   DATA[942,18] := 1.0;
   DATA[942,19] := 1.0;
   DATA[942,20] := 148.808;
   DATA[942,21] := 155.0628;
   DATA[942,22] := 1.71608;
   DATA[942,23] := 928.262;
   DATA[942,24] := 2.0;
   DATA[942,25] := 2.0;
   DATA[942,26] := 7.87798;
   DATA[942,27] := 144.3989;
   DATA[942,28] := 263.0415;
   DATA[942,29] := 11.95847;
   DATA[942,30] := 1.726096;
   DATA[942,31] := 1.281542;
   DATA[942,32] := 0.7357808;
   DATA[942,33] := 0.306761;
   DATA[942,34] := 2.0;
   DATA[942,35] := 250.7049;
   DATA[942,36] := 1.746067;
   DATA[942,37] := 189.5187;
   DATA[942,38] := 0.000128152;
   DATA[942,39] := 1.0;
   DATA[943,0] := 2.542356;
   DATA[943,1] := 627.6909;
   DATA[943,2] := 2.0;
   DATA[943,3] := 1.0;
   DATA[943,4] := 262.4648;
   DATA[943,5] := 8.460844;
   DATA[943,6] := 315.4576;
   DATA[943,8] := 1.0;
   DATA[943,9] := 1.0;
   DATA[943,10] := 1.0;
   DATA[943,11] := 2.010372;
   DATA[943,13] := 1010.839;
   DATA[943,14] := 1.0;
   DATA[943,15] := 1.0;
   DATA[943,16] := 1.0;
   DATA[943,17] := 1.0;
   DATA[943,18] := 1.0;
   DATA[943,19] := 1.0;
   DATA[943,20] := 148.808;
   DATA[943,21] := 155.0628;
   DATA[943,22] := 1.71608;
   DATA[943,23] := 928.1466;
   DATA[943,24] := 2.0;
   DATA[943,25] := 2.0;
   DATA[943,26] := 7.87798;
   DATA[943,27] := 144.3989;
   DATA[943,28] := 263.0415;
   DATA[943,29] := 11.95847;
   DATA[943,30] := 1.726096;
   DATA[943,31] := 1.287306;
   DATA[943,32] := 0.7357808;
   DATA[943,33] := 0.3070813;
   DATA[943,34] := 2.0;
   DATA[943,35] := 250.7049;
   DATA[943,36] := 1.746067;
   DATA[943,37] := 189.5187;
   DATA[943,38] := 0.000128152;
   DATA[943,39] := 1.0;
   DATA[944,0] := 2.540435;
   DATA[944,1] := 627.6124;
   DATA[944,2] := 2.0;
   DATA[944,3] := 1.0;
   DATA[944,4] := 262.4648;
   DATA[944,5] := 8.460844;
   DATA[944,6] := 315.4576;
   DATA[944,8] := 1.0;
   DATA[944,9] := 1.0;
   DATA[944,10] := 1.0;
   DATA[944,11] := 2.010372;
   DATA[944,13] := 1010.718;
   DATA[944,14] := 1.0;
   DATA[944,15] := 1.0;
   DATA[944,16] := 1.0;
   DATA[944,17] := 1.0;
   DATA[944,18] := 1.0;
   DATA[944,19] := 1.0;
   DATA[944,20] := 148.808;
   DATA[944,21] := 155.0628;
   DATA[944,22] := 1.717489;
   DATA[944,23] := 928.1466;
   DATA[944,24] := 2.0;
   DATA[944,25] := 2.0;
   DATA[944,26] := 7.87798;
   DATA[944,27] := 144.3989;
   DATA[944,28] := 263.0415;
   DATA[944,29] := 11.95847;
   DATA[944,30] := 1.728659;
   DATA[944,31] := 1.290893;
   DATA[944,32] := 0.7357808;
   DATA[944,33] := 0.3070813;
   DATA[944,34] := 2.0;
   DATA[944,35] := 250.7049;
   DATA[944,36] := 1.746067;
   DATA[944,37] := 189.5187;
   DATA[944,38] := 0.000128152;
   DATA[944,39] := 1.0;
   DATA[945,0] := 2.540435;
   DATA[945,1] := 627.8086;
   DATA[945,2] := 2.0;
   DATA[945,3] := 1.0;
   DATA[945,4] := 262.4648;
   DATA[945,5] := 8.460844;
   DATA[945,6] := 315.4576;
   DATA[945,8] := 1.0;
   DATA[945,9] := 1.0;
   DATA[945,10] := 1.0;
   DATA[945,11] := 2.010372;
   DATA[945,13] := 1010.959;
   DATA[945,14] := 1.0;
   DATA[945,15] := 1.0;
   DATA[945,16] := 1.0;
   DATA[945,17] := 1.0;
   DATA[945,18] := 1.0;
   DATA[945,19] := 1.0;
   DATA[945,20] := 148.808;
   DATA[945,21] := 155.0628;
   DATA[945,22] := 1.717489;
   DATA[945,23] := 928.1466;
   DATA[945,24] := 2.0;
   DATA[945,25] := 2.0;
   DATA[945,26] := 7.87798;
   DATA[945,27] := 144.3989;
   DATA[945,28] := 263.0415;
   DATA[945,29] := 11.95847;
   DATA[945,30] := 1.728659;
   DATA[945,31] := 1.271551;
   DATA[945,32] := 0.7357808;
   DATA[945,33] := 0.3070813;
   DATA[945,34] := 2.0;
   DATA[945,35] := 250.7049;
   DATA[945,36] := 1.746067;
   DATA[945,37] := 189.5187;
   DATA[945,38] := 0.000128152;
   DATA[945,39] := 1.0;
   DATA[946,0] := 2.540435;
   DATA[946,1] := 628.4366;
   DATA[946,2] := 2.0;
   DATA[946,3] := 1.0;
   DATA[946,4] := 262.4648;
   DATA[946,5] := 8.460844;
   DATA[946,6] := 315.4576;
   DATA[946,8] := 1.0;
   DATA[946,9] := 1.0;
   DATA[946,10] := 1.0;
   DATA[946,11] := 2.010372;
   DATA[946,13] := 1010.638;
   DATA[946,14] := 1.0;
   DATA[946,15] := 1.0;
   DATA[946,16] := 1.0;
   DATA[946,17] := 1.0;
   DATA[946,18] := 1.0;
   DATA[946,19] := 1.0;
   DATA[946,20] := 148.808;
   DATA[946,21] := 155.0628;
   DATA[946,22] := 1.717489;
   DATA[946,23] := 927.8005;
   DATA[946,24] := 2.0;
   DATA[946,25] := 2.0;
   DATA[946,26] := 7.87798;
   DATA[946,27] := 144.3989;
   DATA[946,28] := 263.0415;
   DATA[946,29] := 12.07383;
   DATA[946,30] := 1.728659;
   DATA[946,31] := 1.265275;
   DATA[946,32] := 0.7348846;
   DATA[946,33] := 0.3066329;
   DATA[946,34] := 2.0;
   DATA[946,35] := 250.5608;
   DATA[946,36] := 1.746067;
   DATA[946,37] := 189.5187;
   DATA[946,38] := 0.000128152;
   DATA[946,39] := 1.0;
   DATA[947,0] := 2.545239;
   DATA[947,1] := 629.3395;
   DATA[947,2] := 2.0;
   DATA[947,3] := 1.0;
   DATA[947,4] := 262.4648;
   DATA[947,5] := 8.460844;
   DATA[947,6] := 315.4576;
   DATA[947,8] := 1.0;
   DATA[947,9] := 1.0;
   DATA[947,10] := 1.0;
   DATA[947,11] := 2.010372;
   DATA[947,13] := 1011.119;
   DATA[947,14] := 1.0;
   DATA[947,15] := 1.0;
   DATA[947,16] := 1.0;
   DATA[947,17] := 1.0;
   DATA[947,18] := 1.0;
   DATA[947,19] := 1.0;
   DATA[947,20] := 148.808;
   DATA[947,21] := 155.0628;
   DATA[947,22] := 1.717489;
   DATA[947,23] := 927.3007;
   DATA[947,24] := 2.0;
   DATA[947,25] := 2.0;
   DATA[947,26] := 7.87798;
   DATA[947,27] := 144.3989;
   DATA[947,28] := 263.0415;
   DATA[947,29] := 12.07383;
   DATA[947,30] := 1.728659;
   DATA[947,31] := 1.267196;
   DATA[947,32] := 0.7348846;
   DATA[947,33] := 0.3066329;
   DATA[947,34] := 2.0;
   DATA[947,35] := 250.5447;
   DATA[947,36] := 1.746067;
   DATA[947,37] := 189.5187;
   DATA[947,38] := 0.000128152;
   DATA[947,39] := 1.0;
   DATA[948,0] := 2.552926;
   DATA[948,1] := 630.1245;
   DATA[948,2] := 2.0;
   DATA[948,3] := 1.0;
   DATA[948,4] := 262.4648;
   DATA[948,5] := 8.460844;
   DATA[948,6] := 315.4576;
   DATA[948,8] := 1.0;
   DATA[948,9] := 1.0;
   DATA[948,10] := 1.0;
   DATA[948,11] := 2.010372;
   DATA[948,13] := 1010.638;
   DATA[948,14] := 1.0;
   DATA[948,15] := 1.0;
   DATA[948,16] := 1.0;
   DATA[948,17] := 1.0;
   DATA[948,18] := 1.0;
   DATA[948,19] := 1.0;
   DATA[948,20] := 148.808;
   DATA[948,21] := 155.0628;
   DATA[948,22] := 1.717489;
   DATA[948,23] := 927.1085;
   DATA[948,24] := 2.0;
   DATA[948,25] := 2.0;
   DATA[948,26] := 7.87798;
   DATA[948,27] := 144.3989;
   DATA[948,28] := 263.0415;
   DATA[948,29] := 12.07383;
   DATA[948,30] := 1.728659;
   DATA[948,31] := 1.261176;
   DATA[948,32] := 0.7348846;
   DATA[948,33] := 0.3066329;
   DATA[948,34] := 2.0;
   DATA[948,35] := 250.5447;
   DATA[948,36] := 1.746067;
   DATA[948,37] := 189.3585;
   DATA[948,38] := 0.000128152;
   DATA[948,39] := 1.0;
   DATA[949,0] := 2.55773;
   DATA[949,1] := 631.3414;
   DATA[949,2] := 2.0;
   DATA[949,3] := 1.0;
   DATA[949,4] := 262.4648;
   DATA[949,5] := 8.460844;
   DATA[949,6] := 315.4576;
   DATA[949,8] := 1.0;
   DATA[949,9] := 1.0;
   DATA[949,10] := 1.0;
   DATA[949,11] := 2.010372;
   DATA[949,13] := 1011.159;
   DATA[949,14] := 1.0;
   DATA[949,15] := 1.0;
   DATA[949,16] := 1.0;
   DATA[949,17] := 1.0;
   DATA[949,18] := 1.0;
   DATA[949,19] := 1.0;
   DATA[949,20] := 148.808;
   DATA[949,21] := 155.0628;
   DATA[949,22] := 1.717489;
   DATA[949,23] := 927.3007;
   DATA[949,24] := 2.0;
   DATA[949,25] := 2.0;
   DATA[949,26] := 7.87798;
   DATA[949,27] := 144.3989;
   DATA[949,28] := 263.0415;
   DATA[949,29] := 12.07383;
   DATA[949,30] := 1.728659;
   DATA[949,31] := 1.265659;
   DATA[949,32] := 0.7348846;
   DATA[949,33] := 0.3066329;
   DATA[949,34] := 2.0;
   DATA[949,35] := 250.5447;
   DATA[949,36] := 1.746067;
   DATA[949,37] := 189.3585;
   DATA[949,38] := 0.000128152;
   DATA[949,39] := 1.0;
   DATA[950,0] := 2.55773;
   DATA[950,1] := 632.3619;
   DATA[950,2] := 2.0;
   DATA[950,3] := 1.0;
   DATA[950,4] := 262.4648;
   DATA[950,5] := 8.460844;
   DATA[950,6] := 315.5089;
   DATA[950,8] := 1.0;
   DATA[950,9] := 1.0;
   DATA[950,10] := 1.0;
   DATA[950,11] := 2.010372;
   DATA[950,13] := 1011.119;
   DATA[950,14] := 1.0;
   DATA[950,15] := 1.0;
   DATA[950,16] := 1.0;
   DATA[950,17] := 1.0;
   DATA[950,18] := 1.0;
   DATA[950,19] := 1.0;
   DATA[950,20] := 148.808;
   DATA[950,21] := 155.0628;
   DATA[950,22] := 1.717489;
   DATA[950,23] := 927.2238;
   DATA[950,24] := 2.0;
   DATA[950,25] := 2.0;
   DATA[950,26] := 7.87798;
   DATA[950,27] := 144.3989;
   DATA[950,28] := 263.0415;
   DATA[950,29] := 12.07383;
   DATA[950,30] := 1.728659;
   DATA[950,31] := 1.280517;
   DATA[950,32] := 0.7348846;
   DATA[950,33] := 0.3066329;
   DATA[950,34] := 2.0;
   DATA[950,35] := 250.5447;
   DATA[950,36] := 1.746067;
   DATA[950,37] := 189.3585;
   DATA[950,38] := 0.000128152;
   DATA[950,39] := 1.0;
   DATA[951,0] := 2.55773;
   DATA[951,1] := 633.3825;
   DATA[951,2] := 2.0;
   DATA[951,3] := 1.0;
   DATA[951,4] := 262.4648;
   DATA[951,5] := 8.460844;
   DATA[951,6] := 315.5601;
   DATA[951,8] := 1.0;
   DATA[951,9] := 1.0;
   DATA[951,10] := 1.0;
   DATA[951,11] := 2.010372;
   DATA[951,13] := 1010.758;
   DATA[951,14] := 1.0;
   DATA[951,15] := 1.0;
   DATA[951,16] := 1.0;
   DATA[951,17] := 1.0;
   DATA[951,18] := 1.0;
   DATA[951,19] := 1.0;
   DATA[951,20] := 148.808;
   DATA[951,21] := 155.2166;
   DATA[951,22] := 1.717489;
   DATA[951,23] := 926.6086;
   DATA[951,24] := 2.0;
   DATA[951,25] := 2.0;
   DATA[951,26] := 7.87798;
   DATA[951,27] := 144.3989;
   DATA[951,28] := 263.0415;
   DATA[951,29] := 12.07383;
   DATA[951,30] := 1.726865;
   DATA[951,31] := 1.291405;
   DATA[951,32] := 0.7348846;
   DATA[951,33] := 0.3066329;
   DATA[951,34] := 2.0;
   DATA[951,35] := 250.4166;
   DATA[951,36] := 1.69801;
   DATA[951,37] := 189.2464;
   DATA[951,38] := 0.000128152;
   DATA[951,39] := 1.0;
   DATA[952,0] := 2.556129;
   DATA[952,1] := 634.1675;
   DATA[952,2] := 2.0;
   DATA[952,3] := 1.0;
   DATA[952,4] := 262.4648;
   DATA[952,5] := 8.460844;
   DATA[952,6] := 315.5601;
   DATA[952,8] := 1.0;
   DATA[952,9] := 1.0;
   DATA[952,10] := 1.0;
   DATA[952,11] := 2.010372;
   DATA[952,13] := 1010.879;
   DATA[952,14] := 1.0;
   DATA[952,15] := 1.0;
   DATA[952,16] := 1.0;
   DATA[952,17] := 1.0;
   DATA[952,18] := 1.0;
   DATA[952,19] := 1.0;
   DATA[952,20] := 148.808;
   DATA[952,21] := 155.2166;
   DATA[952,22] := 1.717489;
   DATA[952,23] := 926.0703;
   DATA[952,24] := 2.0;
   DATA[952,25] := 2.0;
   DATA[952,26] := 7.87798;
   DATA[952,27] := 144.3989;
   DATA[952,28] := 263.0415;
   DATA[952,29] := 12.07383;
   DATA[952,30] := 1.726865;
   DATA[952,31] := 1.300884;
   DATA[952,32] := 0.7348846;
   DATA[952,33] := 0.3072094;
   DATA[952,34] := 2.0;
   DATA[952,35] := 250.4166;
   DATA[952,36] := 1.69801;
   DATA[952,37] := 189.2464;
   DATA[952,38] := 0.000128152;
   DATA[952,39] := 1.0;
   DATA[953,0] := 2.547161;
   DATA[953,1] := 635.2667;
   DATA[953,2] := 2.0;
   DATA[953,3] := 1.0;
   DATA[953,4] := 262.4648;
   DATA[953,5] := 8.460844;
   DATA[953,6] := 315.5601;
   DATA[953,8] := 1.0;
   DATA[953,9] := 1.0;
   DATA[953,10] := 1.0;
   DATA[953,11] := 2.010372;
   DATA[953,13] := 1011.079;
   DATA[953,14] := 1.0;
   DATA[953,15] := 1.0;
   DATA[953,16] := 1.0;
   DATA[953,17] := 1.0;
   DATA[953,18] := 1.0;
   DATA[953,19] := 1.0;
   DATA[953,20] := 148.808;
   DATA[953,21] := 155.2166;
   DATA[953,22] := 1.717489;
   DATA[953,23] := 925.6857;
   DATA[953,24] := 2.0;
   DATA[953,25] := 2.0;
   DATA[953,26] := 7.87798;
   DATA[953,27] := 144.3989;
   DATA[953,28] := 263.0415;
   DATA[953,29] := 12.07383;
   DATA[953,30] := 1.726737;
   DATA[953,31] := 1.300243;
   DATA[953,32] := 0.7348846;
   DATA[953,33] := 0.30785;
   DATA[953,34] := 2.0;
   DATA[953,35] := 250.4166;
   DATA[953,36] := 1.69801;
   DATA[953,37] := 189.2464;
   DATA[953,38] := 0.000128152;
   DATA[953,39] := 1.0;
   DATA[954,0] := 2.547161;
   DATA[954,1] := 635.2274;
   DATA[954,2] := 2.0;
   DATA[954,3] := 1.0;
   DATA[954,4] := 262.4648;
   DATA[954,5] := 8.460844;
   DATA[954,6] := 315.6114;
   DATA[954,8] := 1.0;
   DATA[954,9] := 1.0;
   DATA[954,10] := 1.0;
   DATA[954,11] := 2.010372;
   DATA[954,13] := 1010.758;
   DATA[954,14] := 1.0;
   DATA[954,15] := 1.0;
   DATA[954,16] := 1.0;
   DATA[954,17] := 1.0;
   DATA[954,18] := 1.0;
   DATA[954,19] := 1.0;
   DATA[954,20] := 148.808;
   DATA[954,21] := 155.0115;
   DATA[954,22] := 1.717489;
   DATA[954,23] := 925.7626;
   DATA[954,24] := 2.0;
   DATA[954,25] := 2.0;
   DATA[954,26] := 7.87798;
   DATA[954,27] := 144.3989;
   DATA[954,28] := 263.0415;
   DATA[954,29] := 12.07383;
   DATA[954,30] := 1.725968;
   DATA[954,31] := 1.292174;
   DATA[954,32] := 0.7348846;
   DATA[954,33] := 0.3084905;
   DATA[954,34] := 2.0;
   DATA[954,35] := 250.4005;
   DATA[954,36] := 1.69801;
   DATA[954,37] := 189.2464;
   DATA[954,38] := 0.000128152;
   DATA[954,39] := 1.0;
   DATA[955,0] := 2.542677;
   DATA[955,1] := 636.2872;
   DATA[955,2] := 2.0;
   DATA[955,3] := 1.0;
   DATA[955,4] := 262.4648;
   DATA[955,5] := 8.460844;
   DATA[955,6] := 315.6114;
   DATA[955,8] := 1.0;
   DATA[955,9] := 1.0;
   DATA[955,10] := 1.0;
   DATA[955,11] := 2.010372;
   DATA[955,13] := 1010.758;
   DATA[955,14] := 1.0;
   DATA[955,15] := 1.0;
   DATA[955,16] := 1.0;
   DATA[955,17] := 1.0;
   DATA[955,18] := 1.0;
   DATA[955,19] := 1.0;
   DATA[955,20] := 148.808;
   DATA[955,21] := 155.0115;
   DATA[955,22] := 1.717489;
   DATA[955,23] := 925.0705;
   DATA[955,24] := 2.0;
   DATA[955,25] := 2.0;
   DATA[955,26] := 7.87798;
   DATA[955,27] := 144.3989;
   DATA[955,28] := 263.0415;
   DATA[955,29] := 12.07383;
   DATA[955,30] := 1.725583;
   DATA[955,31] := 1.292174;
   DATA[955,32] := 0.7357808;
   DATA[955,33] := 0.3084905;
   DATA[955,34] := 2.0;
   DATA[955,35] := 250.4005;
   DATA[955,36] := 1.69801;
   DATA[955,37] := 189.2464;
   DATA[955,38] := 0.000128152;
   DATA[955,39] := 1.0;
   DATA[956,0] := 2.542677;
   DATA[956,1] := 636.6013;
   DATA[956,2] := 2.0;
   DATA[956,3] := 1.0;
   DATA[956,4] := 262.4648;
   DATA[956,5] := 8.460844;
   DATA[956,6] := 315.6114;
   DATA[956,8] := 1.0;
   DATA[956,9] := 1.0;
   DATA[956,10] := 1.0;
   DATA[956,11] := 2.010372;
   DATA[956,13] := 1010.919;
   DATA[956,14] := 1.0;
   DATA[956,15] := 1.0;
   DATA[956,16] := 1.0;
   DATA[956,17] := 1.0;
   DATA[956,18] := 1.0;
   DATA[956,19] := 1.0;
   DATA[956,20] := 148.808;
   DATA[956,21] := 155.0115;
   DATA[956,22] := 1.714542;
   DATA[956,23] := 924.6475;
   DATA[956,24] := 2.0;
   DATA[956,25] := 2.0;
   DATA[956,26] := 7.87798;
   DATA[956,27] := 144.3989;
   DATA[956,28] := 263.0415;
   DATA[956,29] := 12.07383;
   DATA[956,30] := 1.725583;
   DATA[956,31] := 1.296273;
   DATA[956,32] := 0.7357808;
   DATA[956,33] := 0.3084905;
   DATA[956,34] := 2.0;
   DATA[956,35] := 250.4005;
   DATA[956,36] := 1.69801;
   DATA[956,37] := 189.2464;
   DATA[956,38] := 0.000128152;
   DATA[956,39] := 1.0;
   DATA[957,0] := 2.542677;
   DATA[957,1] := 637.2686;
   DATA[957,2] := 2.0;
   DATA[957,3] := 1.0;
   DATA[957,4] := 262.4648;
   DATA[957,5] := 8.460844;
   DATA[957,6] := 315.6114;
   DATA[957,8] := 1.0;
   DATA[957,9] := 1.0;
   DATA[957,10] := 1.0;
   DATA[957,11] := 2.010372;
   DATA[957,13] := 1010.718;
   DATA[957,14] := 1.0;
   DATA[957,15] := 1.0;
   DATA[957,16] := 1.0;
   DATA[957,17] := 1.0;
   DATA[957,18] := 1.0;
   DATA[957,19] := 1.0;
   DATA[957,20] := 148.808;
   DATA[957,21] := 155.2166;
   DATA[957,22] := 1.714542;
   DATA[957,23] := 924.0707;
   DATA[957,24] := 2.0;
   DATA[957,25] := 2.0;
   DATA[957,26] := 7.87798;
   DATA[957,27] := 144.3989;
   DATA[957,28] := 263.0415;
   DATA[957,29] := 12.07383;
   DATA[957,30] := 1.724045;
   DATA[957,31] := 1.302677;
   DATA[957,32] := 0.7357808;
   DATA[957,33] := 0.3084905;
   DATA[957,34] := 2.0;
   DATA[957,35] := 250.4005;
   DATA[957,36] := 1.69801;
   DATA[957,37] := 189.2464;
   DATA[957,38] := 0.000128152;
   DATA[957,39] := 1.0;
   DATA[958,0] := 2.550364;
   DATA[958,1] := 637.5825;
   DATA[958,2] := 2.0;
   DATA[958,3] := 1.0;
   DATA[958,4] := 262.4648;
   DATA[958,5] := 8.460844;
   DATA[958,6] := 315.6114;
   DATA[958,8] := 1.0;
   DATA[958,9] := 1.0;
   DATA[958,10] := 1.0;
   DATA[958,11] := 2.010372;
   DATA[958,13] := 1010.518;
   DATA[958,14] := 1.0;
   DATA[958,15] := 1.0;
   DATA[958,16] := 1.0;
   DATA[958,17] := 1.0;
   DATA[958,18] := 1.0;
   DATA[958,19] := 1.0;
   DATA[958,20] := 148.808;
   DATA[958,21] := 155.2166;
   DATA[958,22] := 1.714542;
   DATA[958,23] := 923.5709;
   DATA[958,24] := 2.0;
   DATA[958,25] := 2.0;
   DATA[958,26] := 7.87798;
   DATA[958,27] := 144.3989;
   DATA[958,28] := 263.0415;
   DATA[958,29] := 12.07383;
   DATA[958,30] := 1.724045;
   DATA[958,31] := 1.302677;
   DATA[958,32] := 0.7357808;
   DATA[958,33] := 0.3084905;
   DATA[958,34] := 2.0;
   DATA[958,35] := 250.4005;
   DATA[958,36] := 1.69801;
   DATA[958,37] := 189.2464;
   DATA[958,38] := 0.000128152;
   DATA[958,39] := 1.0;
   DATA[959,0] := 2.552285;
   DATA[959,1] := 638.6031;
   DATA[959,2] := 2.0;
   DATA[959,3] := 1.0;
   DATA[959,4] := 262.4648;
   DATA[959,5] := 8.460844;
   DATA[959,6] := 315.6114;
   DATA[959,8] := 1.0;
   DATA[959,9] := 1.0;
   DATA[959,10] := 1.0;
   DATA[959,11] := 2.010372;
   DATA[959,13] := 1010.678;
   DATA[959,14] := 1.0;
   DATA[959,15] := 1.0;
   DATA[959,16] := 1.0;
   DATA[959,17] := 1.0;
   DATA[959,18] := 1.0;
   DATA[959,19] := 1.0;
   DATA[959,20] := 148.808;
   DATA[959,21] := 155.2166;
   DATA[959,22] := 1.715183;
   DATA[959,23] := 923.1479;
   DATA[959,24] := 2.0;
   DATA[959,25] := 2.0;
   DATA[959,26] := 7.87798;
   DATA[959,27] := 144.3989;
   DATA[959,28] := 263.0415;
   DATA[959,29] := 12.07383;
   DATA[959,30] := 1.724045;
   DATA[959,31] := 1.295376;
   DATA[959,32] := 0.7380853;
   DATA[959,33] := 0.3084905;
   DATA[959,34] := 2.0;
   DATA[959,35] := 250.4005;
   DATA[959,36] := 1.69801;
   DATA[959,37] := 189.2464;
   DATA[959,38] := 0.000128152;
   DATA[959,39] := 1.0;
   DATA[960,0] := 2.552285;
   DATA[960,1] := 639.5452;
   DATA[960,2] := 2.0;
   DATA[960,3] := 1.0;
   DATA[960,4] := 262.4648;
   DATA[960,5] := 8.460844;
   DATA[960,6] := 315.6114;
   DATA[960,8] := 1.0;
   DATA[960,9] := 1.0;
   DATA[960,10] := 1.0;
   DATA[960,11] := 2.010372;
   DATA[960,13] := 1010.839;
   DATA[960,14] := 1.0;
   DATA[960,15] := 1.0;
   DATA[960,16] := 1.0;
   DATA[960,17] := 1.0;
   DATA[960,18] := 1.0;
   DATA[960,19] := 1.0;
   DATA[960,20] := 148.808;
   DATA[960,21] := 155.2166;
   DATA[960,22] := 1.71608;
   DATA[960,23] := 922.9941;
   DATA[960,24] := 2.0;
   DATA[960,25] := 2.0;
   DATA[960,26] := 7.87798;
   DATA[960,27] := 144.3989;
   DATA[960,28] := 263.0415;
   DATA[960,29] := 12.07383;
   DATA[960,30] := 1.724045;
   DATA[960,31] := 1.283079;
   DATA[960,32] := 0.7380853;
   DATA[960,33] := 0.3084905;
   DATA[960,34] := 2.0;
   DATA[960,35] := 250.4005;
   DATA[960,36] := 1.69801;
   DATA[960,37] := 189.2464;
   DATA[960,38] := 0.000128152;
   DATA[960,39] := 1.0;
   DATA[961,0] := 2.552285;
   DATA[961,1] := 639.8592;
   DATA[961,2] := 2.0;
   DATA[961,3] := 1.0;
   DATA[961,4] := 262.4648;
   DATA[961,5] := 8.460844;
   DATA[961,6] := 315.6114;
   DATA[961,8] := 1.0;
   DATA[961,9] := 1.0;
   DATA[961,10] := 1.0;
   DATA[961,11] := 2.010372;
   DATA[961,13] := 1011.079;
   DATA[961,14] := 1.0;
   DATA[961,15] := 1.0;
   DATA[961,16] := 1.0;
   DATA[961,17] := 1.0;
   DATA[961,18] := 1.0;
   DATA[961,19] := 1.0;
   DATA[961,20] := 148.808;
   DATA[961,21] := 155.2166;
   DATA[961,22] := 1.71608;
   DATA[961,23] := 922.9172;
   DATA[961,24] := 2.0;
   DATA[961,25] := 2.0;
   DATA[961,26] := 7.87798;
   DATA[961,27] := 144.3989;
   DATA[961,28] := 263.0415;
   DATA[961,29] := 12.07383;
   DATA[961,30] := 1.724045;
   DATA[961,31] := 1.285513;
   DATA[961,32] := 0.7380853;
   DATA[961,33] := 0.3084905;
   DATA[961,34] := 2.0;
   DATA[961,35] := 250.1122;
   DATA[961,36] := 1.746067;
   DATA[961,37] := 189.1022;
   DATA[961,38] := 0.000128152;
   DATA[961,39] := 1.0;
   DATA[962,0] := 2.548762;
   DATA[962,1] := 640.5265;
   DATA[962,2] := 2.0;
   DATA[962,3] := 1.0;
   DATA[962,4] := 262.4648;
   DATA[962,5] := 8.460844;
   DATA[962,6] := 315.6114;
   DATA[962,8] := 1.0;
   DATA[962,9] := 1.0;
   DATA[962,10] := 1.0;
   DATA[962,11] := 2.010372;
   DATA[962,13] := 1010.758;
   DATA[962,14] := 1.0;
   DATA[962,15] := 1.0;
   DATA[962,16] := 1.0;
   DATA[962,17] := 1.0;
   DATA[962,18] := 1.0;
   DATA[962,19] := 1.0;
   DATA[962,20] := 148.808;
   DATA[962,21] := 155.2166;
   DATA[962,22] := 1.714798;
   DATA[962,23] := 922.6096;
   DATA[962,24] := 2.0;
   DATA[962,25] := 2.0;
   DATA[962,26] := 7.87798;
   DATA[962,27] := 144.3989;
   DATA[962,28] := 263.0415;
   DATA[962,29] := 12.07383;
   DATA[962,30] := 1.724045;
   DATA[962,31] := 1.291918;
   DATA[962,32] := 0.7380853;
   DATA[962,33] := 0.3084905;
   DATA[962,34] := 2.0;
   DATA[962,35] := 250.1122;
   DATA[962,36] := 1.762086;
   DATA[962,37] := 189.1022;
   DATA[962,38] := 0.000128152;
   DATA[962,39] := 1.0;
   DATA[963,0] := 2.543317;
   DATA[963,1] := 641.233;
   DATA[963,2] := 2.0;
   DATA[963,3] := 1.0;
   DATA[963,4] := 262.4648;
   DATA[963,5] := 8.462767;
   DATA[963,6] := 315.6114;
   DATA[963,8] := 1.0;
   DATA[963,9] := 1.0;
   DATA[963,10] := 1.0;
   DATA[963,11] := 2.010372;
   DATA[963,13] := 1010.919;
   DATA[963,14] := 1.0;
   DATA[963,15] := 1.0;
   DATA[963,16] := 1.0;
   DATA[963,17] := 1.0;
   DATA[963,18] := 1.0;
   DATA[963,19] := 1.0;
   DATA[963,20] := 148.808;
   DATA[963,21] := 155.1653;
   DATA[963,22] := 1.713261;
   DATA[963,23] := 922.6865;
   DATA[963,24] := 2.0;
   DATA[963,25] := 2.0;
   DATA[963,26] := 7.87798;
   DATA[963,27] := 144.3989;
   DATA[963,28] := 263.0415;
   DATA[963,29] := 12.07383;
   DATA[963,30] := 1.724045;
   DATA[963,31] := 1.30985;
   DATA[963,32] := 0.7380853;
   DATA[963,33] := 0.3084905;
   DATA[963,34] := 2.0;
   DATA[963,35] := 250.1122;
   DATA[963,36] := 1.762086;
   DATA[963,37] := 189.1022;
   DATA[963,38] := 0.000128152;
   DATA[963,39] := 1.0;
   DATA[964,0] := 2.540435;
   DATA[964,1] := 641.5863;
   DATA[964,2] := 2.0;
   DATA[964,3] := 1.0;
   DATA[964,4] := 262.4648;
   DATA[964,5] := 8.463408;
   DATA[964,6] := 315.6114;
   DATA[964,8] := 1.0;
   DATA[964,9] := 1.0;
   DATA[964,10] := 1.0;
   DATA[964,11] := 2.010372;
   DATA[964,13] := 1010.518;
   DATA[964,14] := 1.0;
   DATA[964,15] := 1.0;
   DATA[964,16] := 1.0;
   DATA[964,17] := 1.0;
   DATA[964,18] := 1.0;
   DATA[964,19] := 1.0;
   DATA[964,20] := 148.808;
   DATA[964,21] := 155.1653;
   DATA[964,22] := 1.713261;
   DATA[964,23] := 922.8018;
   DATA[964,24] := 2.0;
   DATA[964,25] := 2.0;
   DATA[964,26] := 7.87798;
   DATA[964,27] := 144.3989;
   DATA[964,28] := 263.0415;
   DATA[964,29] := 12.07383;
   DATA[964,30] := 1.724045;
   DATA[964,31] := 1.307416;
   DATA[964,32] := 0.7380853;
   DATA[964,33] := 0.3084905;
   DATA[964,34] := 2.0;
   DATA[964,35] := 250.1122;
   DATA[964,36] := 1.762086;
   DATA[964,37] := 189.1022;
   DATA[964,38] := 0.000128152;
   DATA[964,39] := 1.0;
   DATA[965,0] := 2.540435;
   DATA[965,1] := 642.1359;
   DATA[965,2] := 2.0;
   DATA[965,3] := 1.0;
   DATA[965,4] := 262.4648;
   DATA[965,5] := 8.463408;
   DATA[965,6] := 315.6114;
   DATA[965,8] := 1.0;
   DATA[965,9] := 1.0;
   DATA[965,10] := 1.0;
   DATA[965,11] := 2.010372;
   DATA[965,13] := 1010.839;
   DATA[965,14] := 1.0;
   DATA[965,15] := 1.0;
   DATA[965,16] := 1.0;
   DATA[965,17] := 1.0;
   DATA[965,18] := 1.0;
   DATA[965,19] := 1.0;
   DATA[965,20] := 148.808;
   DATA[965,21] := 155.1653;
   DATA[965,22] := 1.713261;
   DATA[965,23] := 922.3405;
   DATA[965,24] := 2.0;
   DATA[965,25] := 2.0;
   DATA[965,26] := 7.87798;
   DATA[965,27] := 144.3989;
   DATA[965,28] := 263.0415;
   DATA[965,29] := 12.07383;
   DATA[965,30] := 1.724045;
   DATA[965,31] := 1.302165;
   DATA[965,32] := 0.7380853;
   DATA[965,33] := 0.3084905;
   DATA[965,34] := 2.0;
   DATA[965,35] := 250.1122;
   DATA[965,36] := 1.762086;
   DATA[965,37] := 189.006;
   DATA[965,38] := 0.000128152;
   DATA[965,39] := 1.0;
   DATA[966,0] := 2.540435;
   DATA[966,1] := 642.2929;
   DATA[966,2] := 2.0;
   DATA[966,3] := 1.0;
   DATA[966,4] := 262.4648;
   DATA[966,5] := 8.463408;
   DATA[966,6] := 315.6114;
   DATA[966,8] := 1.0;
   DATA[966,9] := 1.0;
   DATA[966,10] := 1.0;
   DATA[966,11] := 2.010372;
   DATA[966,13] := 1010.558;
   DATA[966,14] := 1.0;
   DATA[966,15] := 1.0;
   DATA[966,16] := 1.0;
   DATA[966,17] := 1.0;
   DATA[966,18] := 1.0;
   DATA[966,19] := 1.0;
   DATA[966,20] := 148.808;
   DATA[966,21] := 155.1653;
   DATA[966,22] := 1.712748;
   DATA[966,23] := 921.8021;
   DATA[966,24] := 2.0;
   DATA[966,25] := 2.0;
   DATA[966,26] := 7.87798;
   DATA[966,27] := 144.3989;
   DATA[966,28] := 263.0415;
   DATA[966,29] := 12.07383;
   DATA[966,30] := 1.723532;
   DATA[966,31] := 1.307801;
   DATA[966,32] := 0.7351407;
   DATA[966,33] := 0.3084905;
   DATA[966,34] := 2.0;
   DATA[966,35] := 250.1122;
   DATA[966,36] := 1.762086;
   DATA[966,37] := 189.006;
   DATA[966,38] := 0.000128152;
   DATA[966,39] := 1.0;
   DATA[967,0] := 2.538513;
   DATA[967,1] := 641.9789;
   DATA[967,2] := 2.0;
   DATA[967,3] := 1.0;
   DATA[967,4] := 262.4648;
   DATA[967,5] := 8.463408;
   DATA[967,6] := 315.6114;
   DATA[967,8] := 1.0;
   DATA[967,9] := 1.0;
   DATA[967,10] := 1.0;
   DATA[967,11] := 2.010372;
   DATA[967,13] := 1010.919;
   DATA[967,14] := 1.0;
   DATA[967,15] := 1.0;
   DATA[967,16] := 1.0;
   DATA[967,17] := 1.0;
   DATA[967,18] := 1.0;
   DATA[967,19] := 1.0;
   DATA[967,20] := 148.808;
   DATA[967,21] := 155.1653;
   DATA[967,22] := 1.712748;
   DATA[967,23] := 921.8021;
   DATA[967,24] := 2.0;
   DATA[967,25] := 2.0;
   DATA[967,26] := 7.87798;
   DATA[967,27] := 144.3989;
   DATA[967,28] := 263.0415;
   DATA[967,29] := 12.07383;
   DATA[967,30] := 1.723532;
   DATA[967,31] := 1.302165;
   DATA[967,32] := 0.7351407;
   DATA[967,33] := 0.3084905;
   DATA[967,34] := 2.0;
   DATA[967,35] := 250.1122;
   DATA[967,36] := 1.762086;
   DATA[967,37] := 188.9419;
   DATA[967,38] := 0.000128152;
   DATA[967,39] := 1.0;
   DATA[968,0] := 2.538513;
   DATA[968,1] := 641.7433;
   DATA[968,2] := 2.0;
   DATA[968,3] := 1.0;
   DATA[968,4] := 262.4648;
   DATA[968,5] := 8.463408;
   DATA[968,6] := 315.6114;
   DATA[968,8] := 1.0;
   DATA[968,9] := 1.0;
   DATA[968,10] := 1.0;
   DATA[968,11] := 2.010372;
   DATA[968,13] := 1010.919;
   DATA[968,14] := 1.0;
   DATA[968,15] := 1.0;
   DATA[968,16] := 1.0;
   DATA[968,17] := 1.0;
   DATA[968,18] := 1.0;
   DATA[968,19] := 1.0;
   DATA[968,20] := 148.808;
   DATA[968,21] := 155.1653;
   DATA[968,22] := 1.712748;
   DATA[968,23] := 921.1484;
   DATA[968,24] := 2.0;
   DATA[968,25] := 2.0;
   DATA[968,26] := 7.87798;
   DATA[968,27] := 144.3989;
   DATA[968,28] := 263.0415;
   DATA[968,29] := 12.07383;
   DATA[968,30] := 1.723532;
   DATA[968,31] := 1.3005;
   DATA[968,32] := 0.7351407;
   DATA[968,33] := 0.3084905;
   DATA[968,34] := 2.0;
   DATA[968,35] := 250.1122;
   DATA[968,36] := 1.762086;
   DATA[968,37] := 188.9419;
   DATA[968,38] := 0.000128152;
   DATA[968,39] := 1.0;
   DATA[969,0] := 2.548442;
   DATA[969,1] := 641.7041;
   DATA[969,2] := 2.0;
   DATA[969,3] := 1.0;
   DATA[969,4] := 262.4648;
   DATA[969,5] := 8.463408;
   DATA[969,6] := 315.6114;
   DATA[969,8] := 1.0;
   DATA[969,9] := 1.0;
   DATA[969,10] := 1.0;
   DATA[969,11] := 2.010372;
   DATA[969,13] := 1011.279;
   DATA[969,14] := 1.0;
   DATA[969,15] := 1.0;
   DATA[969,16] := 1.0;
   DATA[969,17] := 1.0;
   DATA[969,18] := 1.0;
   DATA[969,19] := 1.0;
   DATA[969,20] := 148.808;
   DATA[969,21] := 155.1653;
   DATA[969,22] := 1.714286;
   DATA[969,23] := 921.0331;
   DATA[969,24] := 2.0;
   DATA[969,25] := 2.0;
   DATA[969,26] := 7.87798;
   DATA[969,27] := 144.3989;
   DATA[969,28] := 263.0415;
   DATA[969,29] := 12.07383;
   DATA[969,30] := 1.723532;
   DATA[969,31] := 1.309082;
   DATA[969,32] := 0.7351407;
   DATA[969,33] := 0.3084905;
   DATA[969,34] := 2.0;
   DATA[969,35] := 250.1122;
   DATA[969,36] := 1.762086;
   DATA[969,37] := 188.9419;
   DATA[969,38] := 0.000128152;
   DATA[969,39] := 1.0;
   DATA[970,0] := 2.549082;
   DATA[970,1] := 641.1938;
   DATA[970,2] := 2.0;
   DATA[970,3] := 1.0;
   DATA[970,4] := 262.4648;
   DATA[970,5] := 8.463408;
   DATA[970,6] := 315.637;
   DATA[970,8] := 1.0;
   DATA[970,9] := 1.0;
   DATA[970,10] := 1.0;
   DATA[970,11] := 2.010372;
   DATA[970,13] := 1010.919;
   DATA[970,14] := 1.0;
   DATA[970,15] := 1.0;
   DATA[970,16] := 1.0;
   DATA[970,17] := 1.0;
   DATA[970,18] := 1.0;
   DATA[970,19] := 1.0;
   DATA[970,20] := 148.808;
   DATA[970,21] := 155.1653;
   DATA[970,22] := 1.715567;
   DATA[970,23] := 920.3794;
   DATA[970,24] := 2.0;
   DATA[970,25] := 2.0;
   DATA[970,26] := 7.87798;
   DATA[970,27] := 144.3989;
   DATA[970,28] := 263.0415;
   DATA[970,29] := 12.07383;
   DATA[970,30] := 1.723532;
   DATA[970,31] := 1.305367;
   DATA[970,32] := 0.7351407;
   DATA[970,33] := 0.3084905;
   DATA[970,34] := 2.0;
   DATA[970,35] := 250.1122;
   DATA[970,36] := 1.665972;
   DATA[970,37] := 188.9419;
   DATA[970,38] := 0.000128152;
   DATA[970,39] := 1.0;
   DATA[971,0] := 2.552926;
   DATA[971,1] := 641.3508;
   DATA[971,2] := 2.0;
   DATA[971,3] := 1.0;
   DATA[971,4] := 262.4648;
   DATA[971,5] := 8.463408;
   DATA[971,6] := 315.7396;
   DATA[971,8] := 1.0;
   DATA[971,9] := 1.0;
   DATA[971,10] := 1.0;
   DATA[971,11] := 2.010372;
   DATA[971,13] := 1010.839;
   DATA[971,14] := 1.0;
   DATA[971,15] := 1.0;
   DATA[971,16] := 1.0;
   DATA[971,17] := 1.0;
   DATA[971,18] := 1.0;
   DATA[971,19] := 1.0;
   DATA[971,20] := 148.808;
   DATA[971,21] := 155.1653;
   DATA[971,22] := 1.71608;
   DATA[971,23] := 919.9949;
   DATA[971,24] := 2.0;
   DATA[971,25] := 2.0;
   DATA[971,26] := 7.87798;
   DATA[971,27] := 144.3989;
   DATA[971,28] := 263.0415;
   DATA[971,29] := 12.07383;
   DATA[971,30] := 1.723661;
   DATA[971,31] := 1.309082;
   DATA[971,32] := 0.7351407;
   DATA[971,33] := 0.3084905;
   DATA[971,34] := 2.0;
   DATA[971,35] := 250.4005;
   DATA[971,36] := 1.665972;
   DATA[971,37] := 189.3425;
   DATA[971,38] := 0.000128152;
   DATA[971,39] := 1.0;
   DATA[972,0] := 2.555168;
   DATA[972,1] := 641.7041;
   DATA[972,2] := 2.0;
   DATA[972,3] := 1.0;
   DATA[972,4] := 262.4648;
   DATA[972,5] := 8.463408;
   DATA[972,6] := 315.7396;
   DATA[972,8] := 1.0;
   DATA[972,9] := 1.0;
   DATA[972,10] := 1.0;
   DATA[972,11] := 2.010372;
   DATA[972,13] := 1010.879;
   DATA[972,14] := 1.0;
   DATA[972,15] := 1.0;
   DATA[972,16] := 1.0;
   DATA[972,17] := 1.0;
   DATA[972,18] := 1.0;
   DATA[972,19] := 1.0;
   DATA[972,20] := 148.808;
   DATA[972,21] := 155.1653;
   DATA[972,22] := 1.717361;
   DATA[972,23] := 919.6488;
   DATA[972,24] := 2.0;
   DATA[972,25] := 2.0;
   DATA[972,26] := 7.87798;
   DATA[972,27] := 144.3989;
   DATA[972,28] := 263.0415;
   DATA[972,29] := 12.07383;
   DATA[972,30] := 1.725583;
   DATA[972,31] := 1.312284;
   DATA[972,32] := 0.7351407;
   DATA[972,33] := 0.3083624;
   DATA[972,34] := 2.0;
   DATA[972,35] := 250.4166;
   DATA[972,36] := 1.665972;
   DATA[972,37] := 189.3425;
   DATA[972,38] := 0.000128152;
   DATA[972,39] := 1.0;
   DATA[973,0] := 2.555168;
   DATA[973,1] := 642.1359;
   DATA[973,2] := 2.0;
   DATA[973,3] := 1.0;
   DATA[973,4] := 262.4648;
   DATA[973,5] := 8.463408;
   DATA[973,6] := 315.7396;
   DATA[973,8] := 1.0;
   DATA[973,9] := 1.0;
   DATA[973,10] := 1.0;
   DATA[973,11] := 2.010372;
   DATA[973,13] := 1011.039;
   DATA[973,14] := 1.0;
   DATA[973,15] := 1.0;
   DATA[973,16] := 1.0;
   DATA[973,17] := 1.0;
   DATA[973,18] := 1.0;
   DATA[973,19] := 1.0;
   DATA[973,20] := 148.808;
   DATA[973,21] := 155.1653;
   DATA[973,22] := 1.718515;
   DATA[973,23] := 919.4181;
   DATA[973,24] := 2.0;
   DATA[973,25] := 2.0;
   DATA[973,26] := 7.87798;
   DATA[973,27] := 144.3989;
   DATA[973,28] := 263.0415;
   DATA[973,29] := 12.07383;
   DATA[973,30] := 1.726096;
   DATA[973,31] := 1.303318;
   DATA[973,32] := 0.7351407;
   DATA[973,33] := 0.3083624;
   DATA[973,34] := 2.0;
   DATA[973,35] := 250.5447;
   DATA[973,36] := 1.665972;
   DATA[973,37] := 189.3425;
   DATA[973,38] := 0.000128152;
   DATA[973,39] := 1.0;
   DATA[974,0] := 2.555168;
   DATA[974,1] := 641.9789;
   DATA[974,2] := 2.0;
   DATA[974,3] := 1.0;
   DATA[974,4] := 262.4648;
   DATA[974,5] := 8.463408;
   DATA[974,6] := 315.7396;
   DATA[974,8] := 1.0;
   DATA[974,9] := 1.0;
   DATA[974,10] := 1.0;
   DATA[974,11] := 2.010372;
   DATA[974,13] := 1011.079;
   DATA[974,14] := 1.0;
   DATA[974,15] := 1.0;
   DATA[974,16] := 1.0;
   DATA[974,17] := 1.0;
   DATA[974,18] := 1.0;
   DATA[974,19] := 1.0;
   DATA[974,20] := 148.808;
   DATA[974,21] := 155.1653;
   DATA[974,22] := 1.718515;
   DATA[974,23] := 919.1105;
   DATA[974,24] := 2.0;
   DATA[974,25] := 2.0;
   DATA[974,26] := 7.87798;
   DATA[974,27] := 144.3989;
   DATA[974,28] := 263.0415;
   DATA[974,29] := 12.07383;
   DATA[974,30] := 1.726096;
   DATA[974,31] := 1.288971;
   DATA[974,32] := 0.7351407;
   DATA[974,33] := 0.3083624;
   DATA[974,34] := 2.0;
   DATA[974,35] := 250.5928;
   DATA[974,36] := 1.69801;
   DATA[974,37] := 189.3425;
   DATA[974,38] := 0.000128152;
   DATA[974,39] := 1.0;
   DATA[975,0] := 2.550684;
   DATA[975,1] := 643.392;
   DATA[975,2] := 2.0;
   DATA[975,3] := 1.0;
   DATA[975,4] := 262.4648;
   DATA[975,5] := 8.463408;
   DATA[975,6] := 315.7396;
   DATA[975,8] := 1.0;
   DATA[975,9] := 1.0;
   DATA[975,10] := 1.0;
   DATA[975,11] := 2.010372;
   DATA[975,13] := 1010.839;
   DATA[975,14] := 1.0;
   DATA[975,15] := 1.0;
   DATA[975,16] := 1.0;
   DATA[975,17] := 1.0;
   DATA[975,18] := 1.0;
   DATA[975,19] := 1.0;
   DATA[975,20] := 148.808;
   DATA[975,21] := 155.1653;
   DATA[975,22] := 1.718515;
   DATA[975,23] := 918.8413;
   DATA[975,24] := 2.0;
   DATA[975,25] := 2.0;
   DATA[975,26] := 7.87798;
   DATA[975,27] := 144.3989;
   DATA[975,28] := 263.0415;
   DATA[975,29] := 12.07383;
   DATA[975,30] := 1.726096;
   DATA[975,31] := 1.281542;
   DATA[975,32] := 0.7351407;
   DATA[975,33] := 0.3083624;
   DATA[975,34] := 2.0;
   DATA[975,35] := 250.5928;
   DATA[975,36] := 1.730048;
   DATA[975,37] := 189.3425;
   DATA[975,38] := 0.000128152;
   DATA[975,39] := 1.0;
   DATA[976,0] := 2.548442;
   DATA[976,1] := 644.2555;
   DATA[976,2] := 2.0;
   DATA[976,3] := 1.0;
   DATA[976,4] := 262.4648;
   DATA[976,5] := 8.464369;
   DATA[976,6] := 315.7396;
   DATA[976,8] := 1.0;
   DATA[976,9] := 1.0;
   DATA[976,10] := 1.0;
   DATA[976,11] := 2.010372;
   DATA[976,13] := 1011.079;
   DATA[976,14] := 1.0;
   DATA[976,15] := 1.0;
   DATA[976,16] := 1.0;
   DATA[976,17] := 1.0;
   DATA[976,18] := 1.0;
   DATA[976,19] := 1.0;
   DATA[976,20] := 148.808;
   DATA[976,21] := 155.1653;
   DATA[976,22] := 1.718515;
   DATA[976,23] := 918.5337;
   DATA[976,24] := 2.0;
   DATA[976,25] := 2.0;
   DATA[976,26] := 7.87798;
   DATA[976,27] := 144.3989;
   DATA[976,28] := 263.0415;
   DATA[976,29] := 12.07383;
   DATA[976,30] := 1.725455;
   DATA[976,31] := 1.281542;
   DATA[976,32] := 0.7351407;
   DATA[976,33] := 0.3083624;
   DATA[976,34] := 2.0;
   DATA[976,35] := 250.5928;
   DATA[976,36] := 1.730048;
   DATA[976,37] := 189.3425;
   DATA[976,38] := 0.000128152;
   DATA[976,39] := 1.0;
   DATA[977,0] := 2.538833;
   DATA[977,1] := 645.1191;
   DATA[977,2] := 2.0;
   DATA[977,3] := 1.0;
   DATA[977,4] := 262.4648;
   DATA[977,5] := 8.464369;
   DATA[977,6] := 315.6883;
   DATA[977,8] := 1.0;
   DATA[977,9] := 1.0;
   DATA[977,10] := 1.0;
   DATA[977,11] := 2.010372;
   DATA[977,13] := 1011.159;
   DATA[977,14] := 1.0;
   DATA[977,15] := 1.0;
   DATA[977,16] := 1.0;
   DATA[977,17] := 1.0;
   DATA[977,18] := 1.0;
   DATA[977,19] := 1.0;
   DATA[977,20] := 148.808;
   DATA[977,21] := 155.1653;
   DATA[977,22] := 1.718515;
   DATA[977,23] := 918.1107;
   DATA[977,24] := 2.0;
   DATA[977,25] := 2.0;
   DATA[977,26] := 7.87798;
   DATA[977,27] := 144.3989;
   DATA[977,28] := 263.0415;
   DATA[977,29] := 12.07383;
   DATA[977,30] := 1.725455;
   DATA[977,31] := 1.271935;
   DATA[977,32] := 0.7351407;
   DATA[977,33] := 0.3083624;
   DATA[977,34] := 2.0;
   DATA[977,35] := 250.5928;
   DATA[977,36] := 1.730048;
   DATA[977,37] := 189.3425;
   DATA[977,38] := 0.000128152;
   DATA[977,39] := 1.0;
   DATA[978,0] := 2.536912;
   DATA[978,1] := 646.5322;
   DATA[978,2] := 2.0;
   DATA[978,3] := 1.0;
   DATA[978,4] := 262.4648;
   DATA[978,5] := 8.464369;
   DATA[978,6] := 315.6883;
   DATA[978,8] := 1.0;
   DATA[978,9] := 1.0;
   DATA[978,10] := 1.0;
   DATA[978,11] := 2.010372;
   DATA[978,13] := 1011.119;
   DATA[978,14] := 1.0;
   DATA[978,15] := 1.0;
   DATA[978,16] := 1.0;
   DATA[978,17] := 1.0;
   DATA[978,18] := 1.0;
   DATA[978,19] := 1.0;
   DATA[978,20] := 148.808;
   DATA[978,21] := 155.1653;
   DATA[978,22] := 1.716592;
   DATA[978,23] := 917.9185;
   DATA[978,24] := 2.0;
   DATA[978,25] := 2.0;
   DATA[978,26] := 7.87798;
   DATA[978,27] := 144.3989;
   DATA[978,28] := 263.0415;
   DATA[978,29] := 12.07383;
   DATA[978,30] := 1.725455;
   DATA[978,31] := 1.271679;
   DATA[978,32] := 0.7351407;
   DATA[978,33] := 0.3083624;
   DATA[978,34] := 2.0;
   DATA[978,35] := 250.5928;
   DATA[978,36] := 1.730048;
   DATA[978,37] := 189.3425;
   DATA[978,38] := 0.000128152;
   DATA[978,39] := 1.0;
   DATA[979,0] := 2.535951;
   DATA[979,1] := 647.8275;
   DATA[979,2] := 2.0;
   DATA[979,3] := 1.0;
   DATA[979,4] := 262.4648;
   DATA[979,5] := 8.464369;
   DATA[979,6] := 315.6883;
   DATA[979,8] := 1.0;
   DATA[979,9] := 1.0;
   DATA[979,10] := 1.0;
   DATA[979,11] := 2.010372;
   DATA[979,13] := 1011.439;
   DATA[979,14] := 1.0;
   DATA[979,15] := 1.0;
   DATA[979,16] := 1.0;
   DATA[979,17] := 1.0;
   DATA[979,18] := 1.0;
   DATA[979,19] := 1.0;
   DATA[979,20] := 148.808;
   DATA[979,21] := 155.1653;
   DATA[979,22] := 1.716592;
   DATA[979,23] := 917.6108;
   DATA[979,24] := 2.0;
   DATA[979,25] := 2.0;
   DATA[979,26] := 7.87798;
   DATA[979,27] := 144.3989;
   DATA[979,28] := 263.0415;
   DATA[979,29] := 12.07383;
   DATA[979,30] := 1.725968;
   DATA[979,31] := 1.276419;
   DATA[979,32] := 0.7351407;
   DATA[979,33] := 0.3083624;
   DATA[979,34] := 2.0;
   DATA[979,35] := 250.5928;
   DATA[979,36] := 1.730048;
   DATA[979,37] := 189.3425;
   DATA[979,38] := 0.000128152;
   DATA[979,39] := 1.0;
   DATA[980,0] := 2.535951;
   DATA[980,1] := 647.8275;
   DATA[980,2] := 2.0;
   DATA[980,3] := 1.0;
   DATA[980,4] := 262.4648;
   DATA[980,5] := 8.464369;
   DATA[980,6] := 315.6883;
   DATA[980,8] := 1.0;
   DATA[980,9] := 1.0;
   DATA[980,10] := 1.0;
   DATA[980,11] := 2.010372;
   DATA[980,13] := 1011.439;
   DATA[980,14] := 1.0;
   DATA[980,15] := 1.0;
   DATA[980,16] := 1.0;
   DATA[980,17] := 1.0;
   DATA[980,18] := 1.0;
   DATA[980,19] := 1.0;
   DATA[980,20] := 148.808;
   DATA[980,21] := 155.1653;
   DATA[980,22] := 1.716592;
   DATA[980,23] := 917.6108;
   DATA[980,24] := 2.0;
   DATA[980,25] := 2.0;
   DATA[980,26] := 7.87798;
   DATA[980,27] := 144.3989;
   DATA[980,28] := 263.0415;
   DATA[980,29] := 12.07383;
   DATA[980,30] := 1.725968;
   DATA[980,31] := 1.276419;
   DATA[980,32] := 0.7351407;
   DATA[980,33] := 0.3083624;
   DATA[980,34] := 2.0;
   DATA[980,35] := 250.5928;
   DATA[980,36] := 1.730048;
   DATA[980,37] := 189.3425;
   DATA[980,38] := 0.000128152;
   DATA[980,39] := 1.0;
   DATA[981,0] := 2.533709;
   DATA[981,1] := 648.2985;
   DATA[981,2] := 2.0;
   DATA[981,3] := 1.0;
   DATA[981,4] := 262.4648;
   DATA[981,5] := 8.464369;
   DATA[981,6] := 315.6883;
   DATA[981,8] := 1.0;
   DATA[981,9] := 1.0;
   DATA[981,10] := 1.0;
   DATA[981,11] := 2.010372;
   DATA[981,13] := 1010.839;
   DATA[981,14] := 1.0;
   DATA[981,15] := 1.0;
   DATA[981,16] := 1.0;
   DATA[981,17] := 1.0;
   DATA[981,18] := 1.0;
   DATA[981,19] := 1.0;
   DATA[981,20] := 148.808;
   DATA[981,21] := 155.1653;
   DATA[981,22] := 1.716592;
   DATA[981,23] := 916.9572;
   DATA[981,24] := 2.0;
   DATA[981,25] := 2.0;
   DATA[981,26] := 7.87798;
   DATA[981,27] := 144.3989;
   DATA[981,28] := 263.0415;
   DATA[981,29] := 12.07383;
   DATA[981,30] := 1.726993;
   DATA[981,31] := 1.276419;
   DATA[981,32] := 0.7351407;
   DATA[981,33] := 0.306761;
   DATA[981,34] := 2.0;
   DATA[981,35] := 250.5928;
   DATA[981,36] := 1.730048;
   DATA[981,37] := 189.3425;
   DATA[981,38] := 0.000128152;
   DATA[981,39] := 1.0;
   DATA[982,0] := 2.534029;
   DATA[982,1] := 648.7696;
   DATA[982,2] := 2.0;
   DATA[982,3] := 1.0;
   DATA[982,4] := 262.4648;
   DATA[982,5] := 8.464369;
   DATA[982,6] := 315.6883;
   DATA[982,8] := 1.0;
   DATA[982,9] := 1.0;
   DATA[982,10] := 1.0;
   DATA[982,11] := 2.010372;
   DATA[982,13] := 1010.919;
   DATA[982,14] := 1.0;
   DATA[982,15] := 1.0;
   DATA[982,16] := 1.0;
   DATA[982,17] := 1.0;
   DATA[982,18] := 1.0;
   DATA[982,19] := 1.0;
   DATA[982,20] := 148.808;
   DATA[982,21] := 155.1653;
   DATA[982,22] := 1.714542;
   DATA[982,23] := 916.7265;
   DATA[982,24] := 2.0;
   DATA[982,25] := 2.0;
   DATA[982,26] := 7.87798;
   DATA[982,27] := 144.3989;
   DATA[982,28] := 263.1056;
   DATA[982,29] := 12.07383;
   DATA[982,30] := 1.726993;
   DATA[982,31] := 1.281158;
   DATA[982,32] := 0.7351407;
   DATA[982,33] := 0.306761;
   DATA[982,34] := 2.0;
   DATA[982,35] := 250.5928;
   DATA[982,36] := 1.730048;
   DATA[982,37] := 189.3425;
   DATA[982,38] := 0.000128152;
   DATA[982,39] := 1.0;
   DATA[983,0] := 2.540755;
   DATA[983,1] := 649.3584;
   DATA[983,2] := 2.0;
   DATA[983,3] := 1.0;
   DATA[983,4] := 262.4648;
   DATA[983,5] := 8.464369;
   DATA[983,6] := 315.6883;
   DATA[983,8] := 1.0;
   DATA[983,9] := 1.0;
   DATA[983,10] := 1.0;
   DATA[983,11] := 2.010372;
   DATA[983,13] := 1010.879;
   DATA[983,14] := 1.0;
   DATA[983,15] := 1.0;
   DATA[983,16] := 1.0;
   DATA[983,17] := 1.0;
   DATA[983,18] := 1.0;
   DATA[983,19] := 1.0;
   DATA[983,20] := 148.808;
   DATA[983,21] := 155.1653;
   DATA[983,22] := 1.712748;
   DATA[983,23] := 916.342;
   DATA[983,24] := 2.0;
   DATA[983,25] := 2.0;
   DATA[983,26] := 7.87798;
   DATA[983,27] := 144.3989;
   DATA[983,28] := 263.1056;
   DATA[983,29] := 12.07383;
   DATA[983,30] := 1.726993;
   DATA[983,31] := 1.282183;
   DATA[983,32] := 0.7351407;
   DATA[983,33] := 0.306761;
   DATA[983,34] := 2.0;
   DATA[983,35] := 250.4967;
   DATA[983,36] := 1.730048;
   DATA[983,37] := 189.3425;
   DATA[983,38] := 0.000128152;
   DATA[983,39] := 1.0;
   DATA[984,0] := 2.54684;
   DATA[984,1] := 650.2612;
   DATA[984,2] := 2.0;
   DATA[984,3] := 1.0;
   DATA[984,4] := 262.4648;
   DATA[984,5] := 8.464369;
   DATA[984,6] := 315.6883;
   DATA[984,8] := 1.0;
   DATA[984,9] := 1.0;
   DATA[984,10] := 1.0;
   DATA[984,11] := 2.010372;
   DATA[984,13] := 1010.678;
   DATA[984,14] := 1.0;
   DATA[984,15] := 1.0;
   DATA[984,16] := 1.0;
   DATA[984,17] := 1.0;
   DATA[984,18] := 1.0;
   DATA[984,19] := 1.0;
   DATA[984,20] := 148.808;
   DATA[984,21] := 155.1653;
   DATA[984,22] := 1.71467;
   DATA[984,23] := 915.6883;
   DATA[984,24] := 2.0;
   DATA[984,25] := 2.0;
   DATA[984,26] := 7.87798;
   DATA[984,27] := 144.3989;
   DATA[984,28] := 263.1056;
   DATA[984,29] := 12.15073;
   DATA[984,30] := 1.726993;
   DATA[984,31] := 1.282183;
   DATA[984,32] := 0.7351407;
   DATA[984,33] := 0.3074016;
   DATA[984,34] := 2.0;
   DATA[984,35] := 250.4326;
   DATA[984,36] := 1.730048;
   DATA[984,37] := 189.3425;
   DATA[984,38] := 0.000128152;
   DATA[984,39] := 1.0;
   DATA[985,0] := 2.551965;
   DATA[985,1] := 650.7715;
   DATA[985,2] := 2.0;
   DATA[985,3] := 1.0;
   DATA[985,4] := 262.4648;
   DATA[985,5] := 8.464369;
   DATA[985,6] := 315.6883;
   DATA[985,8] := 1.0;
   DATA[985,9] := 1.0;
   DATA[985,10] := 1.0;
   DATA[985,11] := 2.010372;
   DATA[985,13] := 1010.678;
   DATA[985,14] := 1.0;
   DATA[985,15] := 1.0;
   DATA[985,16] := 1.0;
   DATA[985,17] := 1.0;
   DATA[985,18] := 1.0;
   DATA[985,19] := 1.0;
   DATA[985,20] := 148.808;
   DATA[985,21] := 155.1653;
   DATA[985,22] := 1.715311;
   DATA[985,23] := 915.4576;
   DATA[985,24] := 2.0;
   DATA[985,25] := 2.0;
   DATA[985,26] := 7.87798;
   DATA[985,27] := 144.3989;
   DATA[985,28] := 263.1056;
   DATA[985,29] := 12.15073;
   DATA[985,30] := 1.726993;
   DATA[985,31] := 1.284104;
   DATA[985,32] := 0.7351407;
   DATA[985,33] := 0.3086186;
   DATA[985,34] := 2.0;
   DATA[985,35] := 250.3845;
   DATA[985,36] := 1.730048;
   DATA[985,37] := 189.3425;
   DATA[985,38] := 0.000128152;
   DATA[985,39] := 1.0;
   DATA[986,0] := 2.551965;
   DATA[986,1] := 651.321;
   DATA[986,2] := 2.0;
   DATA[986,3] := 1.0;
   DATA[986,4] := 262.4648;
   DATA[986,5] := 8.461164;
   DATA[986,6] := 315.6883;
   DATA[986,8] := 1.0;
   DATA[986,9] := 1.0;
   DATA[986,10] := 1.0;
   DATA[986,11] := 2.010372;
   DATA[986,13] := 1010.478;
   DATA[986,14] := 1.0;
   DATA[986,15] := 1.0;
   DATA[986,16] := 1.0;
   DATA[986,17] := 1.0;
   DATA[986,18] := 1.0;
   DATA[986,19] := 1.0;
   DATA[986,20] := 148.808;
   DATA[986,21] := 155.1653;
   DATA[986,22] := 1.717361;
   DATA[986,23] := 915.4191;
   DATA[986,24] := 2.0;
   DATA[986,25] := 2.0;
   DATA[986,26] := 7.87798;
   DATA[986,27] := 144.3989;
   DATA[986,28] := 263.1056;
   DATA[986,29] := 12.15073;
   DATA[986,30] := 1.726993;
   DATA[986,31] := 1.296401;
   DATA[986,32] := 0.7351407;
   DATA[986,33] := 0.3086186;
   DATA[986,34] := 2.0;
   DATA[986,35] := 250.3845;
   DATA[986,36] := 1.730048;
   DATA[986,37] := 189.1182;
   DATA[986,38] := 0.000128152;
   DATA[986,39] := 1.0;
   DATA[987,0] := 2.553886;
   DATA[987,1] := 652.1453;
   DATA[987,2] := 2.0;
   DATA[987,3] := 1.0;
   DATA[987,4] := 262.4648;
   DATA[987,5] := 8.461164;
   DATA[987,6] := 315.6883;
   DATA[987,8] := 1.0;
   DATA[987,9] := 1.0;
   DATA[987,10] := 1.0;
   DATA[987,11] := 2.010372;
   DATA[987,13] := 1010.358;
   DATA[987,14] := 1.0;
   DATA[987,15] := 1.0;
   DATA[987,16] := 1.0;
   DATA[987,17] := 1.0;
   DATA[987,18] := 1.0;
   DATA[987,19] := 1.0;
   DATA[987,20] := 148.808;
   DATA[987,21] := 155.1653;
   DATA[987,22] := 1.718002;
   DATA[987,23] := 914.8423;
   DATA[987,24] := 2.0;
   DATA[987,25] := 2.0;
   DATA[987,26] := 7.87798;
   DATA[987,27] := 144.3989;
   DATA[987,28] := 263.1056;
   DATA[987,29] := 12.15073;
   DATA[987,30] := 1.725711;
   DATA[987,31] := 1.293326;
   DATA[987,32] := 0.7351407;
   DATA[987,33] := 0.3086186;
   DATA[987,34] := 2.0;
   DATA[987,35] := 250.3845;
   DATA[987,36] := 1.730048;
   DATA[987,37] := 189.1182;
   DATA[987,38] := 0.000128152;
   DATA[987,39] := 1.0;
   DATA[988,0] := 2.553886;
   DATA[988,1] := 652.1453;
   DATA[988,2] := 2.0;
   DATA[988,3] := 1.0;
   DATA[988,4] := 262.4648;
   DATA[988,5] := 8.461164;
   DATA[988,6] := 315.6883;
   DATA[988,8] := 1.0;
   DATA[988,9] := 1.0;
   DATA[988,10] := 1.0;
   DATA[988,11] := 2.010372;
   DATA[988,13] := 1010.879;
   DATA[988,14] := 1.0;
   DATA[988,15] := 1.0;
   DATA[988,16] := 1.0;
   DATA[988,17] := 1.0;
   DATA[988,18] := 1.0;
   DATA[988,19] := 1.0;
   DATA[988,20] := 148.808;
   DATA[988,21] := 155.1653;
   DATA[988,22] := 1.718002;
   DATA[988,23] := 914.5347;
   DATA[988,24] := 2.0;
   DATA[988,25] := 2.0;
   DATA[988,26] := 7.87798;
   DATA[988,27] := 144.3989;
   DATA[988,28] := 263.1056;
   DATA[988,29] := 12.15073;
   DATA[988,30] := 1.725327;
   DATA[988,31] := 1.291533;
   DATA[988,32] := 0.7351407;
   DATA[988,33] := 0.3086186;
   DATA[988,34] := 2.0;
   DATA[988,35] := 250.5127;
   DATA[988,36] := 1.730048;
   DATA[988,37] := 189.3585;
   DATA[988,38] := 0.000128152;
   DATA[988,39] := 1.0;
   DATA[989,0] := 2.54684;
   DATA[989,1] := 652.1846;
   DATA[989,2] := 2.0;
   DATA[989,3] := 1.0;
   DATA[989,4] := 262.4648;
   DATA[989,5] := 8.461164;
   DATA[989,6] := 315.6883;
   DATA[989,8] := 1.0;
   DATA[989,9] := 1.0;
   DATA[989,10] := 1.0;
   DATA[989,11] := 2.010372;
   DATA[989,13] := 1010.959;
   DATA[989,14] := 1.0;
   DATA[989,15] := 1.0;
   DATA[989,16] := 1.0;
   DATA[989,17] := 1.0;
   DATA[989,18] := 1.0;
   DATA[989,19] := 1.0;
   DATA[989,20] := 148.808;
   DATA[989,21] := 155.0884;
   DATA[989,22] := 1.719924;
   DATA[989,23] := 914.2271;
   DATA[989,24] := 2.0;
   DATA[989,25] := 2.0;
   DATA[989,26] := 7.87798;
   DATA[989,27] := 144.3989;
   DATA[989,28] := 263.1056;
   DATA[989,29] := 12.15073;
   DATA[989,30] := 1.725327;
   DATA[989,31] := 1.298962;
   DATA[989,32] := 0.7351407;
   DATA[989,33] := 0.3086186;
   DATA[989,34] := 2.0;
   DATA[989,35] := 250.5127;
   DATA[989,36] := 1.730048;
   DATA[989,37] := 189.5668;
   DATA[989,38] := 0.000128152;
   DATA[989,39] := 1.0;
   DATA[990,0] := 2.542036;
   DATA[990,1] := 652.5771;
   DATA[990,2] := 2.0;
   DATA[990,3] := 1.0;
   DATA[990,4] := 262.5288;
   DATA[990,5] := 8.461164;
   DATA[990,6] := 315.7139;
   DATA[990,8] := 1.0;
   DATA[990,9] := 1.0;
   DATA[990,10] := 1.0;
   DATA[990,11] := 2.010372;
   DATA[990,13] := 1010.758;
   DATA[990,14] := 1.0;
   DATA[990,15] := 1.0;
   DATA[990,16] := 1.0;
   DATA[990,17] := 1.0;
   DATA[990,18] := 1.0;
   DATA[990,19] := 1.0;
   DATA[990,20] := 148.808;
   DATA[990,21] := 155.0884;
   DATA[990,22] := 1.719924;
   DATA[990,23] := 913.9195;
   DATA[990,24] := 2.0;
   DATA[990,25] := 2.0;
   DATA[990,26] := 7.87798;
   DATA[990,27] := 144.3989;
   DATA[990,28] := 263.1056;
   DATA[990,29] := 12.15073;
   DATA[990,30] := 1.725327;
   DATA[990,31] := 1.289996;
   DATA[990,32] := 0.7351407;
   DATA[990,33] := 0.3086186;
   DATA[990,34] := 2.0;
   DATA[990,35] := 250.6729;
   DATA[990,36] := 1.730048;
   DATA[990,37] := 189.5668;
   DATA[990,38] := 0.000128152;
   DATA[990,39] := 1.0;
   DATA[991,0] := 2.538513;
   DATA[991,1] := 652.6949;
   DATA[991,2] := 2.0;
   DATA[991,3] := 1.0;
   DATA[991,4] := 262.5288;
   DATA[991,5] := 8.461164;
   DATA[991,6] := 315.8165;
   DATA[991,8] := 1.0;
   DATA[991,9] := 1.0;
   DATA[991,10] := 1.0;
   DATA[991,11] := 2.010372;
   DATA[991,13] := 1010.718;
   DATA[991,14] := 1.0;
   DATA[991,15] := 1.0;
   DATA[991,16] := 1.0;
   DATA[991,17] := 1.0;
   DATA[991,18] := 1.0;
   DATA[991,19] := 1.0;
   DATA[991,20] := 148.808;
   DATA[991,21] := 155.0115;
   DATA[991,22] := 1.719924;
   DATA[991,23] := 913.9964;
   DATA[991,24] := 2.0;
   DATA[991,25] := 2.0;
   DATA[991,26] := 7.87798;
   DATA[991,27] := 144.2707;
   DATA[991,28] := 263.1056;
   DATA[991,29] := 12.15073;
   DATA[991,30] := 1.725327;
   DATA[991,31] := 1.289996;
   DATA[991,32] := 0.7351407;
   DATA[991,33] := 0.3074656;
   DATA[991,34] := 2.0;
   DATA[991,35] := 250.785;
   DATA[991,36] := 1.730048;
   DATA[991,37] := 189.5668;
   DATA[991,38] := 0.000128152;
   DATA[991,39] := 1.0;
   DATA[992,0] := 2.538513;
   DATA[992,1] := 653.1659;
   DATA[992,2] := 2.0;
   DATA[992,3] := 1.0;
   DATA[992,4] := 262.5288;
   DATA[992,5] := 8.461164;
   DATA[992,6] := 315.8165;
   DATA[992,8] := 1.0;
   DATA[992,9] := 1.0;
   DATA[992,10] := 1.0;
   DATA[992,11] := 2.010372;
   DATA[992,13] := 1010.718;
   DATA[992,14] := 1.0;
   DATA[992,15] := 1.0;
   DATA[992,16] := 1.0;
   DATA[992,17] := 1.0;
   DATA[992,18] := 1.0;
   DATA[992,19] := 1.0;
   DATA[992,20] := 148.808;
   DATA[992,21] := 155.0115;
   DATA[992,22] := 1.719924;
   DATA[992,23] := 913.6119;
   DATA[992,24] := 2.0;
   DATA[992,25] := 2.0;
   DATA[992,26] := 7.87798;
   DATA[992,27] := 144.2194;
   DATA[992,28] := 263.1056;
   DATA[992,29] := 12.15073;
   DATA[992,30] := 1.725327;
   DATA[992,31] := 1.290509;
   DATA[992,32] := 0.7351407;
   DATA[992,33] := 0.3066329;
   DATA[992,34] := 2.0;
   DATA[992,35] := 250.785;
   DATA[992,36] := 1.730048;
   DATA[992,37] := 189.5668;
   DATA[992,38] := 0.000128152;
   DATA[992,39] := 1.0;
   DATA[993,0] := 2.538513;
   DATA[993,1] := 653.1659;
   DATA[993,2] := 2.0;
   DATA[993,3] := 1.0;
   DATA[993,4] := 262.5288;
   DATA[993,5] := 8.461164;
   DATA[993,6] := 315.8165;
   DATA[993,8] := 1.0;
   DATA[993,9] := 1.0;
   DATA[993,10] := 1.0;
   DATA[993,11] := 2.010372;
   DATA[993,13] := 1010.678;
   DATA[993,14] := 1.0;
   DATA[993,15] := 1.0;
   DATA[993,16] := 1.0;
   DATA[993,17] := 1.0;
   DATA[993,18] := 1.0;
   DATA[993,19] := 1.0;
   DATA[993,20] := 148.808;
   DATA[993,21] := 155.0115;
   DATA[993,22] := 1.719924;
   DATA[993,23] := 913.3043;
   DATA[993,24] := 2.0;
   DATA[993,25] := 2.0;
   DATA[993,26] := 7.87798;
   DATA[993,27] := 144.2194;
   DATA[993,28] := 263.1056;
   DATA[993,29] := 12.15073;
   DATA[993,30] := 1.727378;
   DATA[993,31] := 1.282183;
   DATA[993,32] := 0.7351407;
   DATA[993,33] := 0.3066329;
   DATA[993,34] := 2.0;
   DATA[993,35] := 250.785;
   DATA[993,36] := 1.730048;
   DATA[993,37] := 189.5668;
   DATA[993,38] := 0.000128152;
   DATA[993,39] := 1.0;
   DATA[994,0] := 2.538513;
   DATA[994,1] := 653.5192;
   DATA[994,2] := 2.0;
   DATA[994,3] := 1.0;
   DATA[994,4] := 262.5288;
   DATA[994,5] := 8.461164;
   DATA[994,6] := 315.8165;
   DATA[994,8] := 1.0;
   DATA[994,9] := 1.0;
   DATA[994,10] := 1.0;
   DATA[994,11] := 2.010372;
   DATA[994,13] := 1010.839;
   DATA[994,14] := 1.0;
   DATA[994,15] := 1.0;
   DATA[994,16] := 1.0;
   DATA[994,17] := 1.0;
   DATA[994,18] := 1.0;
   DATA[994,19] := 1.0;
   DATA[994,20] := 148.808;
   DATA[994,21] := 155.0115;
   DATA[994,22] := 1.720565;
   DATA[994,23] := 912.9197;
   DATA[994,24] := 2.0;
   DATA[994,25] := 2.0;
   DATA[994,26] := 7.87798;
   DATA[994,27] := 144.2194;
   DATA[994,28] := 263.1056;
   DATA[994,29] := 12.15073;
   DATA[994,30] := 1.727378;
   DATA[994,31] := 1.275138;
   DATA[994,32] := 0.7351407;
   DATA[994,33] := 0.3066329;
   DATA[994,34] := 2.0;
   DATA[994,35] := 250.785;
   DATA[994,36] := 1.730048;
   DATA[994,37] := 189.5668;
   DATA[994,38] := 0.000128152;
   DATA[994,39] := 1.0;
   DATA[995,0] := 2.543958;
   DATA[995,1] := 654.3828;
   DATA[995,2] := 2.0;
   DATA[995,3] := 1.0;
   DATA[995,4] := 262.5288;
   DATA[995,5] := 8.461164;
   DATA[995,6] := 315.8165;
   DATA[995,8] := 1.0;
   DATA[995,9] := 1.0;
   DATA[995,10] := 1.0;
   DATA[995,11] := 2.010372;
   DATA[995,13] := 1010.919;
   DATA[995,14] := 1.0;
   DATA[995,15] := 1.0;
   DATA[995,16] := 1.0;
   DATA[995,17] := 1.0;
   DATA[995,18] := 1.0;
   DATA[995,19] := 1.0;
   DATA[995,20] := 148.808;
   DATA[995,21] := 155.0115;
   DATA[995,22] := 1.72095;
   DATA[995,23] := 912.1892;
   DATA[995,24] := 2.0;
   DATA[995,25] := 2.0;
   DATA[995,26] := 7.87798;
   DATA[995,27] := 143.9887;
   DATA[995,28] := 263.1056;
   DATA[995,29] := 12.15073;
   DATA[995,30] := 1.727378;
   DATA[995,31] := 1.264506;
   DATA[995,32] := 0.7351407;
   DATA[995,33] := 0.3066329;
   DATA[995,34] := 2.0;
   DATA[995,35] := 250.785;
   DATA[995,36] := 1.730048;
   DATA[995,37] := 189.5668;
   DATA[995,38] := 0.000128152;
   DATA[995,39] := 1.0;
   DATA[996,0] := 2.548442;
   DATA[996,1] := 654.265;
   DATA[996,2] := 2.0;
   DATA[996,3] := 1.0;
   DATA[996,4] := 262.5288;
   DATA[996,5] := 8.461164;
   DATA[996,6] := 315.8165;
   DATA[996,8] := 1.0;
   DATA[996,9] := 1.0;
   DATA[996,10] := 1.0;
   DATA[996,11] := 2.010372;
   DATA[996,13] := 1011.039;
   DATA[996,14] := 1.0;
   DATA[996,15] := 1.0;
   DATA[996,16] := 1.0;
   DATA[996,17] := 1.0;
   DATA[996,18] := 1.0;
   DATA[996,19] := 1.0;
   DATA[996,20] := 148.808;
   DATA[996,21] := 155.0115;
   DATA[996,22] := 1.719027;
   DATA[996,23] := 911.3817;
   DATA[996,24] := 2.0;
   DATA[996,25] := 2.0;
   DATA[996,26] := 7.87798;
   DATA[996,27] := 143.9887;
   DATA[996,28] := 263.1056;
   DATA[996,29] := 12.15073;
   DATA[996,30] := 1.727378;
   DATA[996,31] := 1.261688;
   DATA[996,32] := 0.7351407;
   DATA[996,33] := 0.3066329;
   DATA[996,34] := 2.0;
   DATA[996,35] := 250.785;
   DATA[996,36] := 1.730048;
   DATA[996,37] := 189.5668;
   DATA[996,38] := 0.000128152;
   DATA[996,39] := 1.0;
   DATA[997,0] := 2.555168;
   DATA[997,1] := 654.7753;
   DATA[997,2] := 2.0;
   DATA[997,3] := 1.0;
   DATA[997,4] := 262.5288;
   DATA[997,5] := 8.461164;
   DATA[997,6] := 315.8165;
   DATA[997,8] := 1.0;
   DATA[997,9] := 1.0;
   DATA[997,10] := 1.0;
   DATA[997,11] := 2.010372;
   DATA[997,13] := 1010.879;
   DATA[997,14] := 1.0;
   DATA[997,15] := 1.0;
   DATA[997,16] := 1.0;
   DATA[997,17] := 1.0;
   DATA[997,18] := 1.0;
   DATA[997,19] := 1.0;
   DATA[997,20] := 148.808;
   DATA[997,21] := 155.0115;
   DATA[997,22] := 1.718515;
   DATA[997,23] := 911.2279;
   DATA[997,24] := 2.0;
   DATA[997,25] := 2.0;
   DATA[997,26] := 7.87798;
   DATA[997,27] := 143.9887;
   DATA[997,28] := 263.1056;
   DATA[997,29] := 12.15073;
   DATA[997,30] := 1.727378;
   DATA[997,31] := 1.27898;
   DATA[997,32] := 0.7351407;
   DATA[997,33] := 0.3066329;
   DATA[997,34] := 2.0;
   DATA[997,35] := 250.785;
   DATA[997,36] := 1.730048;
   DATA[997,37] := 189.5668;
   DATA[997,38] := 0.000128152;
   DATA[997,39] := 1.0;
   DATA[998,0] := 2.555168;
   DATA[998,1] := 655.1285;
   DATA[998,2] := 2.0;
   DATA[998,3] := 1.0;
   DATA[998,4] := 262.5288;
   DATA[998,5] := 8.461164;
   DATA[998,6] := 315.8165;
   DATA[998,8] := 1.0;
   DATA[998,9] := 1.0;
   DATA[998,10] := 1.0;
   DATA[998,11] := 2.010372;
   DATA[998,13] := 1011.239;
   DATA[998,14] := 1.0;
   DATA[998,15] := 1.0;
   DATA[998,16] := 1.0;
   DATA[998,17] := 1.0;
   DATA[998,18] := 1.0;
   DATA[998,19] := 1.0;
   DATA[998,20] := 148.808;
   DATA[998,21] := 155.0115;
   DATA[998,22] := 1.718515;
   DATA[998,23] := 910.9972;
   DATA[998,24] := 2.0;
   DATA[998,25] := 2.0;
   DATA[998,26] := 7.87798;
   DATA[998,27] := 143.9887;
   DATA[998,28] := 263.1056;
   DATA[998,29] := 12.15073;
   DATA[998,30] := 1.727378;
   DATA[998,31] := 1.287947;
   DATA[998,32] := 0.7351407;
   DATA[998,33] := 0.3084265;
   DATA[998,34] := 2.0;
   DATA[998,35] := 250.5608;
   DATA[998,36] := 1.730048;
   DATA[998,37] := 189.4546;
   DATA[998,38] := 0.000128152;
   DATA[998,39] := 1.0;
   DATA[999,0] := 2.55773;
   DATA[999,1] := 655.7173;
   DATA[999,2] := 2.0;
   DATA[999,3] := 1.0;
   DATA[999,4] := 262.5288;
   DATA[999,5] := 8.461164;
   DATA[999,6] := 315.8165;
   DATA[999,8] := 1.0;
   DATA[999,9] := 1.0;
   DATA[999,10] := 1.0;
   DATA[999,11] := 2.010372;
   DATA[999,13] := 1010.839;
   DATA[999,14] := 1.0;
   DATA[999,15] := 1.0;
   DATA[999,16] := 1.0;
   DATA[999,17] := 1.0;
   DATA[999,18] := 1.0;
   DATA[999,19] := 1.0;
   DATA[999,20] := 148.808;
   DATA[999,21] := 155.0115;
   DATA[999,22] := 1.717105;
   DATA[999,23] := 910.7665;
   DATA[999,24] := 2.0;
   DATA[999,25] := 2.0;
   DATA[999,26] := 7.87798;
   DATA[999,27] := 144.2451;
   DATA[999,28] := 263.1056;
   DATA[999,29] := 12.15073;
   DATA[999,30] := 1.727378;
   DATA[999,31] := 1.282567;
   DATA[999,32] := 0.7351407;
   DATA[999,33] := 0.3084265;
   DATA[999,34] := 2.0;
   DATA[999,35] := 250.4967;
   DATA[999,36] := 1.730048;
   DATA[999,37] := 189.4546;
   DATA[999,38] := 0.000128152;
   DATA[999,39] := 1.0;
   DATA[1000,0] := 2.559331;
   DATA[1000,1] := 655.9528;
   DATA[1000,2] := 2.0;
   DATA[1000,3] := 1.0;
   DATA[1000,4] := 262.5288;
   DATA[1000,5] := 8.461164;
   DATA[1000,6] := 315.8165;
   DATA[1000,8] := 1.0;
   DATA[1000,9] := 1.0;
   DATA[1000,10] := 1.0;
   DATA[1000,11] := 2.010372;
   DATA[1000,13] := 1011.159;
   DATA[1000,14] := 1.0;
   DATA[1000,15] := 1.0;
   DATA[1000,16] := 1.0;
   DATA[1000,17] := 1.0;
   DATA[1000,18] := 1.0;
   DATA[1000,19] := 1.0;
   DATA[1000,20] := 148.808;
   DATA[1000,21] := 155.0115;
   DATA[1000,22] := 1.717105;
   DATA[1000,23] := 910.1512;
   DATA[1000,24] := 2.0;
   DATA[1000,25] := 2.0;
   DATA[1000,26] := 7.87798;
   DATA[1000,27] := 144.2451;
   DATA[1000,28] := 263.1056;
   DATA[1000,29] := 12.15073;
   DATA[1000,30] := 1.728659;
   DATA[1000,31] := 1.281798;
   DATA[1000,32] := 0.7351407;
   DATA[1000,33] := 0.3084265;
   DATA[1000,34] := 2.0;
   DATA[1000,35] := 250.4967;
   DATA[1000,36] := 1.730048;
   DATA[1000,37] := 189.4546;
   DATA[1000,38] := 0.000128152;
   DATA[1000,39] := 1.0;
   DATA[1001,0] := 2.550684;
   DATA[1001,1] := 656.5024;
   DATA[1001,2] := 2.0;
   DATA[1001,3] := 1.0;
   DATA[1001,4] := 262.5288;
   DATA[1001,5] := 8.461164;
   DATA[1001,6] := 315.8165;
   DATA[1001,8] := 1.0;
   DATA[1001,9] := 1.0;
   DATA[1001,10] := 1.0;
   DATA[1001,11] := 2.010372;
   DATA[1001,13] := 1010.758;
   DATA[1001,14] := 1.0;
   DATA[1001,15] := 1.0;
   DATA[1001,16] := 1.0;
   DATA[1001,17] := 1.0;
   DATA[1001,18] := 1.0;
   DATA[1001,19] := 1.0;
   DATA[1001,20] := 148.808;
   DATA[1001,21] := 155.0115;
   DATA[1001,22] := 1.717105;
   DATA[1001,23] := 909.8821;
   DATA[1001,24] := 2.0;
   DATA[1001,25] := 2.0;
   DATA[1001,26] := 7.87798;
   DATA[1001,27] := 144.2451;
   DATA[1001,28] := 263.1056;
   DATA[1001,29] := 12.11228;
   DATA[1001,30] := 1.728659;
   DATA[1001,31] := 1.281798;
   DATA[1001,32] := 0.7351407;
   DATA[1001,33] := 0.3084265;
   DATA[1001,34] := 2.0;
   DATA[1001,35] := 250.4967;
   DATA[1001,36] := 1.730048;
   DATA[1001,37] := 189.3265;
   DATA[1001,38] := 0.000128152;
   DATA[1001,39] := 1.0;
   DATA[1002,0] := 2.547161;
   DATA[1002,1] := 656.8164;
   DATA[1002,2] := 2.0;
   DATA[1002,3] := 1.0;
   DATA[1002,4] := 262.5288;
   DATA[1002,5] := 8.462126;
   DATA[1002,6] := 316.0728;
   DATA[1002,8] := 1.0;
   DATA[1002,9] := 1.0;
   DATA[1002,10] := 1.0;
   DATA[1002,11] := 2.010372;
   DATA[1002,13] := 1010.879;
   DATA[1002,14] := 1.0;
   DATA[1002,15] := 1.0;
   DATA[1002,16] := 1.0;
   DATA[1002,17] := 1.0;
   DATA[1002,18] := 1.0;
   DATA[1002,19] := 1.0;
   DATA[1002,20] := 148.808;
   DATA[1002,21] := 155.0115;
   DATA[1002,22] := 1.717105;
   DATA[1002,23] := 909.3822;
   DATA[1002,24] := 2.0;
   DATA[1002,25] := 2.0;
   DATA[1002,26] := 7.87798;
   DATA[1002,27] := 144.2451;
   DATA[1002,28] := 263.1056;
   DATA[1002,29] := 12.11228;
   DATA[1002,30] := 1.728659;
   DATA[1002,31] := 1.281798;
   DATA[1002,32] := 0.7351407;
   DATA[1002,33] := 0.3069532;
   DATA[1002,34] := 2.0;
   DATA[1002,35] := 250.4967;
   DATA[1002,36] := 1.730048;
   DATA[1002,37] := 189.3265;
   DATA[1002,38] := 0.000128152;
   DATA[1002,39] := 1.0;
   DATA[1003,0] := 2.539474;
   DATA[1003,1] := 657.1304;
   DATA[1003,2] := 2.0;
   DATA[1003,3] := 1.0;
   DATA[1003,4] := 262.5288;
   DATA[1003,5] := 8.462126;
   DATA[1003,6] := 316.0728;
   DATA[1003,8] := 1.0;
   DATA[1003,9] := 1.0;
   DATA[1003,10] := 1.0;
   DATA[1003,11] := 2.010372;
   DATA[1003,13] := 1010.959;
   DATA[1003,14] := 1.0;
   DATA[1003,15] := 1.0;
   DATA[1003,16] := 1.0;
   DATA[1003,17] := 1.0;
   DATA[1003,18] := 1.0;
   DATA[1003,19] := 1.0;
   DATA[1003,20] := 148.808;
   DATA[1003,21] := 155.0115;
   DATA[1003,22] := 1.717105;
   DATA[1003,23] := 909.0746;
   DATA[1003,24] := 2.0;
   DATA[1003,25] := 2.0;
   DATA[1003,26] := 7.87798;
   DATA[1003,27] := 144.2451;
   DATA[1003,28] := 263.1056;
   DATA[1003,29] := 12.11228;
   DATA[1003,30] := 1.728531;
   DATA[1003,31] := 1.298834;
   DATA[1003,32] := 0.7351407;
   DATA[1003,33] := 0.3074016;
   DATA[1003,34] := 2.0;
   DATA[1003,35] := 250.4967;
   DATA[1003,36] := 1.730048;
   DATA[1003,37] := 189.2143;
   DATA[1003,38] := 0.000128152;
   DATA[1003,39] := 1.0;
   DATA[1004,0] := 2.536912;
   DATA[1004,1] := 657.4445;
   DATA[1004,2] := 2.0;
   DATA[1004,3] := 1.0;
   DATA[1004,4] := 262.5288;
   DATA[1004,5] := 8.462126;
   DATA[1004,6] := 316.0728;
   DATA[1004,8] := 1.0;
   DATA[1004,9] := 1.0;
   DATA[1004,10] := 1.0;
   DATA[1004,11] := 2.010372;
   DATA[1004,13] := 1011.039;
   DATA[1004,14] := 1.0;
   DATA[1004,15] := 1.0;
   DATA[1004,16] := 1.0;
   DATA[1004,17] := 1.0;
   DATA[1004,18] := 1.0;
   DATA[1004,19] := 1.0;
   DATA[1004,20] := 148.808;
   DATA[1004,21] := 155.0115;
   DATA[1004,22] := 1.717105;
   DATA[1004,23] := 908.8054;
   DATA[1004,24] := 2.0;
   DATA[1004,25] := 2.0;
   DATA[1004,26] := 7.87798;
   DATA[1004,27] := 144.2194;
   DATA[1004,28] := 263.1056;
   DATA[1004,29] := 12.11228;
   DATA[1004,30] := 1.726096;
   DATA[1004,31] := 1.302037;
   DATA[1004,32] := 0.7351407;
   DATA[1004,33] := 0.3077859;
   DATA[1004,34] := 2.0;
   DATA[1004,35] := 250.4967;
   DATA[1004,36] := 1.730048;
   DATA[1004,37] := 189.2143;
   DATA[1004,38] := 0.000128152;
   DATA[1004,39] := 1.0;
   DATA[1005,0] := 2.536271;
   DATA[1005,1] := 658.0725;
   DATA[1005,2] := 2.0;
   DATA[1005,3] := 1.0;
   DATA[1005,4] := 262.5288;
   DATA[1005,5] := 8.462126;
   DATA[1005,6] := 315.8421;
   DATA[1005,8] := 1.0;
   DATA[1005,9] := 1.0;
   DATA[1005,10] := 1.0;
   DATA[1005,11] := 2.010372;
   DATA[1005,13] := 1010.879;
   DATA[1005,14] := 1.0;
   DATA[1005,15] := 1.0;
   DATA[1005,16] := 1.0;
   DATA[1005,17] := 1.0;
   DATA[1005,18] := 1.0;
   DATA[1005,19] := 1.0;
   DATA[1005,20] := 148.808;
   DATA[1005,21] := 155.0115;
   DATA[1005,22] := 1.717105;
   DATA[1005,23] := 908.2671;
   DATA[1005,24] := 2.0;
   DATA[1005,25] := 2.0;
   DATA[1005,26] := 7.87798;
   DATA[1005,27] := 144.0656;
   DATA[1005,28] := 263.1056;
   DATA[1005,29] := 12.11228;
   DATA[1005,30] := 1.726096;
   DATA[1005,31] := 1.292814;
   DATA[1005,32] := 0.7351407;
   DATA[1005,33] := 0.3071454;
   DATA[1005,34] := 2.0;
   DATA[1005,35] := 250.3365;
   DATA[1005,36] := 1.730048;
   DATA[1005,37] := 189.2143;
   DATA[1005,38] := 0.000128152;
   DATA[1005,39] := 1.0;
   DATA[1006,0] := 2.535951;
   DATA[1006,1] := 658.5828;
   DATA[1006,2] := 2.0;
   DATA[1006,3] := 1.0;
   DATA[1006,4] := 262.5288;
   DATA[1006,5] := 8.462126;
   DATA[1006,6] := 315.8421;
   DATA[1006,8] := 1.0;
   DATA[1006,9] := 1.0;
   DATA[1006,10] := 1.0;
   DATA[1006,11] := 2.010372;
   DATA[1006,13] := 1010.558;
   DATA[1006,14] := 1.0;
   DATA[1006,15] := 1.0;
   DATA[1006,16] := 1.0;
   DATA[1006,17] := 1.0;
   DATA[1006,18] := 1.0;
   DATA[1006,19] := 1.0;
   DATA[1006,20] := 148.808;
   DATA[1006,21] := 155.0115;
   DATA[1006,22] := 1.717105;
   DATA[1006,23] := 908.0364;
   DATA[1006,24] := 2.0;
   DATA[1006,25] := 2.0;
   DATA[1006,26] := 7.87798;
   DATA[1006,27] := 144.0656;
   DATA[1006,28] := 263.1056;
   DATA[1006,29] := 12.11228;
   DATA[1006,30] := 1.726096;
   DATA[1006,31] := 1.292046;
   DATA[1006,32] := 0.7351407;
   DATA[1006,33] := 0.3069532;
   DATA[1006,34] := 2.0;
   DATA[1006,35] := 250.3365;
   DATA[1006,36] := 1.730048;
   DATA[1006,37] := 189.2143;
   DATA[1006,38] := 0.000128152;
   DATA[1006,39] := 1.0;
   DATA[1007,0] := 2.535951;
   DATA[1007,1] := 659.2893;
   DATA[1007,2] := 2.0;
   DATA[1007,3] := 1.0;
   DATA[1007,4] := 262.5288;
   DATA[1007,5] := 8.462126;
   DATA[1007,6] := 315.8421;
   DATA[1007,8] := 1.0;
   DATA[1007,9] := 1.0;
   DATA[1007,10] := 1.0;
   DATA[1007,11] := 2.010372;
   DATA[1007,13] := 1010.879;
   DATA[1007,14] := 1.0;
   DATA[1007,15] := 1.0;
   DATA[1007,16] := 1.0;
   DATA[1007,17] := 1.0;
   DATA[1007,18] := 1.0;
   DATA[1007,19] := 1.0;
   DATA[1007,20] := 148.808;
   DATA[1007,21] := 155.0115;
   DATA[1007,22] := 1.717105;
   DATA[1007,23] := 907.6519;
   DATA[1007,24] := 2.0;
   DATA[1007,25] := 2.0;
   DATA[1007,26] := 7.87798;
   DATA[1007,27] := 144.0656;
   DATA[1007,28] := 263.1056;
   DATA[1007,29] := 12.11228;
   DATA[1007,30] := 1.726096;
   DATA[1007,31] := 1.308185;
   DATA[1007,32] := 0.7351407;
   DATA[1007,33] := 0.3072735;
   DATA[1007,34] := 2.0;
   DATA[1007,35] := 250.3365;
   DATA[1007,36] := 1.730048;
   DATA[1007,37] := 189.2143;
   DATA[1007,38] := 0.000128152;
   DATA[1007,39] := 1.0;
   DATA[1008,0] := 2.537232;
   DATA[1008,1] := 659.9566;
   DATA[1008,2] := 2.0;
   DATA[1008,3] := 1.0;
   DATA[1008,4] := 262.5288;
   DATA[1008,5] := 8.462126;
   DATA[1008,6] := 315.8421;
   DATA[1008,8] := 1.0;
   DATA[1008,9] := 1.0;
   DATA[1008,10] := 1.0;
   DATA[1008,11] := 2.010372;
   DATA[1008,13] := 1010.959;
   DATA[1008,14] := 1.0;
   DATA[1008,15] := 1.0;
   DATA[1008,16] := 1.0;
   DATA[1008,17] := 1.0;
   DATA[1008,18] := 1.0;
   DATA[1008,19] := 1.0;
   DATA[1008,20] := 148.808;
   DATA[1008,21] := 155.0115;
   DATA[1008,22] := 1.717105;
   DATA[1008,23] := 907.5365;
   DATA[1008,24] := 2.0;
   DATA[1008,25] := 2.0;
   DATA[1008,26] := 7.87798;
   DATA[1008,27] := 144.0656;
   DATA[1008,28] := 263.1056;
   DATA[1008,29] := 12.11228;
   DATA[1008,30] := 1.727378;
   DATA[1008,31] := 1.311003;
   DATA[1008,32] := 0.7351407;
   DATA[1008,33] := 0.3088108;
   DATA[1008,34] := 2.0;
   DATA[1008,35] := 250.3365;
   DATA[1008,36] := 1.730048;
   DATA[1008,37] := 189.2143;
   DATA[1008,38] := 0.000128152;
   DATA[1008,39] := 1.0;
   DATA[1009,0] := 2.54652;
   DATA[1009,1] := 660.0744;
   DATA[1009,2] := 2.0;
   DATA[1009,3] := 1.0;
   DATA[1009,4] := 262.5288;
   DATA[1009,5] := 8.462126;
   DATA[1009,6] := 315.8421;
   DATA[1009,8] := 1.0;
   DATA[1009,9] := 1.0;
   DATA[1009,10] := 1.0;
   DATA[1009,11] := 2.010372;
   DATA[1009,13] := 1011.239;
   DATA[1009,14] := 1.0;
   DATA[1009,15] := 1.0;
   DATA[1009,16] := 1.0;
   DATA[1009,17] := 1.0;
   DATA[1009,18] := 1.0;
   DATA[1009,19] := 1.0;
   DATA[1009,20] := 148.808;
   DATA[1009,21] := 155.0115;
   DATA[1009,22] := 1.717105;
   DATA[1009,23] := 907.1905;
   DATA[1009,24] := 2.0;
   DATA[1009,25] := 2.0;
   DATA[1009,26] := 7.87798;
   DATA[1009,27] := 144.0656;
   DATA[1009,28] := 263.1056;
   DATA[1009,29] := 12.11228;
   DATA[1009,30] := 1.727378;
   DATA[1009,31] := 1.295376;
   DATA[1009,32] := 0.7351407;
   DATA[1009,33] := 0.3088108;
   DATA[1009,34] := 2.0;
   DATA[1009,35] := 250.3365;
   DATA[1009,36] := 1.649953;
   DATA[1009,37] := 189.2143;
   DATA[1009,38] := 0.000128152;
   DATA[1009,39] := 1.0;
   DATA[1010,0] := 2.551965;
   DATA[1010,1] := 660.0744;
   DATA[1010,2] := 2.0;
   DATA[1010,3] := 1.0;
   DATA[1010,4] := 262.5288;
   DATA[1010,5] := 8.462126;
   DATA[1010,6] := 315.8421;
   DATA[1010,8] := 1.0;
   DATA[1010,9] := 1.0;
   DATA[1010,10] := 1.0;
   DATA[1010,11] := 2.010372;
   DATA[1010,13] := 1010.959;
   DATA[1010,14] := 1.0;
   DATA[1010,15] := 1.0;
   DATA[1010,16] := 1.0;
   DATA[1010,17] := 1.0;
   DATA[1010,18] := 1.0;
   DATA[1010,19] := 1.0;
   DATA[1010,20] := 148.808;
   DATA[1010,21] := 155.0115;
   DATA[1010,22] := 1.717105;
   DATA[1010,23] := 907.2674;
   DATA[1010,24] := 2.0;
   DATA[1010,25] := 2.0;
   DATA[1010,26] := 7.87798;
   DATA[1010,27] := 144.0656;
   DATA[1010,28] := 263.1056;
   DATA[1010,29] := 12.11228;
   DATA[1010,30] := 1.727378;
   DATA[1010,31] := 1.280646;
   DATA[1010,32] := 0.7351407;
   DATA[1010,33] := 0.3088108;
   DATA[1010,34] := 2.0;
   DATA[1010,35] := 250.3365;
   DATA[1010,36] := 1.649953;
   DATA[1010,37] := 189.2143;
   DATA[1010,38] := 0.000128152;
   DATA[1010,39] := 1.0;
   DATA[1011,0] := 2.556129;
   DATA[1011,1] := 661.0164;
   DATA[1011,2] := 2.0;
   DATA[1011,3] := 1.0;
   DATA[1011,4] := 262.5288;
   DATA[1011,5] := 8.462126;
   DATA[1011,6] := 315.8421;
   DATA[1011,8] := 1.0;
   DATA[1011,9] := 1.0;
   DATA[1011,10] := 1.0;
   DATA[1011,11] := 2.010372;
   DATA[1011,13] := 1011.279;
   DATA[1011,14] := 1.0;
   DATA[1011,15] := 1.0;
   DATA[1011,16] := 1.0;
   DATA[1011,17] := 1.0;
   DATA[1011,18] := 1.0;
   DATA[1011,19] := 1.0;
   DATA[1011,20] := 148.808;
   DATA[1011,21] := 155.0115;
   DATA[1011,22] := 1.717105;
   DATA[1011,23] := 906.9213;
   DATA[1011,24] := 2.0;
   DATA[1011,25] := 2.0;
   DATA[1011,26] := 7.87798;
   DATA[1011,27] := 144.0656;
   DATA[1011,28] := 263.1056;
   DATA[1011,29] := 12.11228;
   DATA[1011,30] := 1.727378;
   DATA[1011,31] := 1.261944;
   DATA[1011,32] := 0.7351407;
   DATA[1011,33] := 0.3077859;
   DATA[1011,34] := 2.0;
   DATA[1011,35] := 250.3365;
   DATA[1011,36] := 1.649953;
   DATA[1011,37] := 189.1983;
   DATA[1011,38] := 0.000128152;
   DATA[1011,39] := 1.0;
   DATA[1012,0] := 2.556129;
   DATA[1012,1] := 661.6445;
   DATA[1012,2] := 2.0;
   DATA[1012,3] := 1.0;
   DATA[1012,4] := 262.5288;
   DATA[1012,5] := 8.462126;
   DATA[1012,6] := 315.8421;
   DATA[1012,8] := 1.0;
   DATA[1012,9] := 1.0;
   DATA[1012,10] := 1.0;
   DATA[1012,11] := 2.010372;
   DATA[1012,13] := 1011.079;
   DATA[1012,14] := 1.0;
   DATA[1012,15] := 1.0;
   DATA[1012,16] := 1.0;
   DATA[1012,17] := 1.0;
   DATA[1012,18] := 1.0;
   DATA[1012,19] := 1.0;
   DATA[1012,20] := 148.808;
   DATA[1012,21] := 155.0115;
   DATA[1012,22] := 1.717105;
   DATA[1012,23] := 906.806;
   DATA[1012,24] := 2.0;
   DATA[1012,25] := 2.0;
   DATA[1012,26] := 7.87798;
   DATA[1012,27] := 144.2194;
   DATA[1012,28] := 263.1056;
   DATA[1012,29] := 12.11228;
   DATA[1012,30] := 1.727378;
   DATA[1012,31] := 1.2549;
   DATA[1012,32] := 0.7351407;
   DATA[1012,33] := 0.3077859;
   DATA[1012,34] := 2.0;
   DATA[1012,35] := 250.3365;
   DATA[1012,36] := 1.649953;
   DATA[1012,37] := 189.1983;
   DATA[1012,38] := 0.000128152;
   DATA[1012,39] := 1.0;
   DATA[1013,0] := 2.556129;
   DATA[1013,1] := 662.4296;
   DATA[1013,2] := 2.0;
   DATA[1013,3] := 1.0;
   DATA[1013,4] := 262.5288;
   DATA[1013,5] := 8.462126;
   DATA[1013,6] := 315.8421;
   DATA[1013,8] := 1.0;
   DATA[1013,9] := 1.0;
   DATA[1013,10] := 1.0;
   DATA[1013,11] := 2.010372;
   DATA[1013,13] := 1011.359;
   DATA[1013,14] := 1.0;
   DATA[1013,15] := 1.0;
   DATA[1013,16] := 1.0;
   DATA[1013,17] := 1.0;
   DATA[1013,18] := 1.0;
   DATA[1013,19] := 1.0;
   DATA[1013,20] := 148.808;
   DATA[1013,21] := 155.0115;
   DATA[1013,22] := 1.717105;
   DATA[1013,23] := 906.3445;
   DATA[1013,24] := 2.0;
   DATA[1013,25] := 2.0;
   DATA[1013,26] := 7.87798;
   DATA[1013,27] := 144.2194;
   DATA[1013,28] := 263.1056;
   DATA[1013,29] := 12.11228;
   DATA[1013,30] := 1.724686;
   DATA[1013,31] := 1.254515;
   DATA[1013,32] := 0.7351407;
   DATA[1013,33] := 0.3083624;
   DATA[1013,34] := 2.0;
   DATA[1013,35] := 250.3365;
   DATA[1013,36] := 1.649953;
   DATA[1013,37] := 189.1182;
   DATA[1013,38] := 0.000128152;
   DATA[1013,39] := 1.0;
   DATA[1014,0] := 2.551324;
   DATA[1014,1] := 662.9398;
   DATA[1014,2] := 2.0;
   DATA[1014,3] := 1.0;
   DATA[1014,4] := 262.5288;
   DATA[1014,5] := 8.462126;
   DATA[1014,6] := 315.8421;
   DATA[1014,8] := 1.0;
   DATA[1014,9] := 1.0;
   DATA[1014,10] := 1.0;
   DATA[1014,11] := 2.010372;
   DATA[1014,13] := 1010.839;
   DATA[1014,14] := 1.0;
   DATA[1014,15] := 1.0;
   DATA[1014,16] := 1.0;
   DATA[1014,17] := 1.0;
   DATA[1014,18] := 1.0;
   DATA[1014,19] := 1.0;
   DATA[1014,20] := 148.808;
   DATA[1014,21] := 155.0115;
   DATA[1014,22] := 1.717105;
   DATA[1014,23] := 905.9985;
   DATA[1014,24] := 2.0;
   DATA[1014,25] := 2.0;
   DATA[1014,26] := 7.87798;
   DATA[1014,27] := 144.2194;
   DATA[1014,28] := 263.1056;
   DATA[1014,29] := 12.11228;
   DATA[1014,30] := 1.72443;
   DATA[1014,31] := 1.255284;
   DATA[1014,32] := 0.7351407;
   DATA[1014,33] := 0.3083624;
   DATA[1014,34] := 2.0;
   DATA[1014,35] := 250.3365;
   DATA[1014,36] := 1.649953;
   DATA[1014,37] := 189.1182;
   DATA[1014,38] := 0.000128152;
   DATA[1014,39] := 1.0;
   DATA[1015,0] := 2.551324;
   DATA[1015,1] := 663.1754;
   DATA[1015,2] := 2.0;
   DATA[1015,3] := 1.0;
   DATA[1015,4] := 262.5288;
   DATA[1015,5] := 8.462126;
   DATA[1015,6] := 315.8421;
   DATA[1015,8] := 1.0;
   DATA[1015,9] := 1.0;
   DATA[1015,10] := 1.0;
   DATA[1015,11] := 2.010372;
   DATA[1015,13] := 1010.879;
   DATA[1015,14] := 1.0;
   DATA[1015,15] := 1.0;
   DATA[1015,16] := 1.0;
   DATA[1015,17] := 1.0;
   DATA[1015,18] := 1.0;
   DATA[1015,19] := 1.0;
   DATA[1015,20] := 148.808;
   DATA[1015,21] := 155.0115;
   DATA[1015,22] := 1.717105;
   DATA[1015,23] := 905.8447;
   DATA[1015,24] := 2.0;
   DATA[1015,25] := 2.0;
   DATA[1015,26] := 7.87798;
   DATA[1015,27] := 144.2194;
   DATA[1015,28] := 263.1056;
   DATA[1015,29] := 12.11228;
   DATA[1015,30] := 1.72443;
   DATA[1015,31] := 1.270655;
   DATA[1015,32] := 0.7351407;
   DATA[1015,33] := 0.3083624;
   DATA[1015,34] := 2.0;
   DATA[1015,35] := 250.2403;
   DATA[1015,36] := 1.649953;
   DATA[1015,37] := 189.1182;
   DATA[1015,38] := 0.000128152;
   DATA[1015,39] := 1.0;
   DATA[1016,0] := 2.544919;
   DATA[1016,1] := 663.6856;
   DATA[1016,2] := 2.0;
   DATA[1016,3] := 1.0;
   DATA[1016,4] := 262.5288;
   DATA[1016,5] := 8.462126;
   DATA[1016,6] := 315.9959;
   DATA[1016,8] := 1.0;
   DATA[1016,9] := 1.0;
   DATA[1016,10] := 1.0;
   DATA[1016,11] := 2.010372;
   DATA[1016,13] := 1011.039;
   DATA[1016,14] := 1.0;
   DATA[1016,15] := 1.0;
   DATA[1016,16] := 1.0;
   DATA[1016,17] := 1.0;
   DATA[1016,18] := 1.0;
   DATA[1016,19] := 1.0;
   DATA[1016,20] := 148.808;
   DATA[1016,21] := 155.0115;
   DATA[1016,22] := 1.717105;
   DATA[1016,23] := 905.537;
   DATA[1016,24] := 2.0;
   DATA[1016,25] := 2.0;
   DATA[1016,26] := 7.87798;
   DATA[1016,27] := 144.2194;
   DATA[1016,28] := 263.1056;
   DATA[1016,29] := 12.03538;
   DATA[1016,30] := 1.72443;
   DATA[1016,31] := 1.271935;
   DATA[1016,32] := 0.7351407;
   DATA[1016,33] := 0.3083624;
   DATA[1016,34] := 2.0;
   DATA[1016,35] := 250.2243;
   DATA[1016,36] := 1.649953;
   DATA[1016,37] := 189.1182;
   DATA[1016,38] := 0.000128152;
   DATA[1016,39] := 1.0;
   DATA[1017,0] := 2.541075;
   DATA[1017,1] := 663.8034;
   DATA[1017,2] := 2.0;
   DATA[1017,3] := 1.0;
   DATA[1017,4] := 262.5288;
   DATA[1017,5] := 8.462126;
   DATA[1017,6] := 315.9959;
   DATA[1017,8] := 1.0;
   DATA[1017,9] := 1.0;
   DATA[1017,10] := 1.0;
   DATA[1017,11] := 2.010372;
   DATA[1017,13] := 1011.039;
   DATA[1017,14] := 1.0;
   DATA[1017,15] := 1.0;
   DATA[1017,16] := 1.0;
   DATA[1017,17] := 1.0;
   DATA[1017,18] := 1.0;
   DATA[1017,19] := 1.0;
   DATA[1017,20] := 148.808;
   DATA[1017,21] := 155.0115;
   DATA[1017,22] := 1.715567;
   DATA[1017,23] := 905.2294;
   DATA[1017,24] := 2.0;
   DATA[1017,25] := 2.0;
   DATA[1017,26] := 7.87798;
   DATA[1017,27] := 144.2194;
   DATA[1017,28] := 263.1056;
   DATA[1017,29] := 12.03538;
   DATA[1017,30] := 1.72443;
   DATA[1017,31] := 1.266812;
   DATA[1017,32] := 0.7351407;
   DATA[1017,33] := 0.3083624;
   DATA[1017,34] := 2.0;
   DATA[1017,35] := 250.1442;
   DATA[1017,36] := 1.649953;
   DATA[1017,37] := 189.1182;
   DATA[1017,38] := 0.000128152;
   DATA[1017,39] := 1.0;
   DATA[1018,0] := 2.541075;
   DATA[1018,1] := 664.3137;
   DATA[1018,2] := 2.0;
   DATA[1018,3] := 1.0;
   DATA[1018,4] := 262.5288;
   DATA[1018,5] := 8.462126;
   DATA[1018,6] := 315.9959;
   DATA[1018,8] := 1.0;
   DATA[1018,9] := 1.0;
   DATA[1018,10] := 1.0;
   DATA[1018,11] := 2.010372;
   DATA[1018,13] := 1011.119;
   DATA[1018,14] := 1.0;
   DATA[1018,15] := 1.0;
   DATA[1018,16] := 1.0;
   DATA[1018,17] := 1.0;
   DATA[1018,18] := 1.0;
   DATA[1018,19] := 1.0;
   DATA[1018,20] := 148.808;
   DATA[1018,21] := 155.0115;
   DATA[1018,22] := 1.715567;
   DATA[1018,23] := 905.2679;
   DATA[1018,24] := 2.0;
   DATA[1018,25] := 2.0;
   DATA[1018,26] := 7.87798;
   DATA[1018,27] := 144.1169;
   DATA[1018,28] := 263.1056;
   DATA[1018,29] := 12.03538;
   DATA[1018,30] := 1.72443;
   DATA[1018,31] := 1.268093;
   DATA[1018,32] := 0.7351407;
   DATA[1018,33] := 0.3083624;
   DATA[1018,34] := 2.0;
   DATA[1018,35] := 250.1442;
   DATA[1018,36] := 1.649953;
   DATA[1018,37] := 189.1022;
   DATA[1018,38] := 0.000128152;
   DATA[1018,39] := 1.0;
   DATA[1019,0] := 2.541075;
   DATA[1019,1] := 664.7062;
   DATA[1019,2] := 2.0;
   DATA[1019,3] := 1.0;
   DATA[1019,4] := 262.5288;
   DATA[1019,5] := 8.462126;
   DATA[1019,6] := 315.9959;
   DATA[1019,8] := 1.0;
   DATA[1019,9] := 1.0;
   DATA[1019,10] := 1.0;
   DATA[1019,11] := 2.010372;
   DATA[1019,13] := 1011.439;
   DATA[1019,14] := 1.0;
   DATA[1019,15] := 1.0;
   DATA[1019,16] := 1.0;
   DATA[1019,17] := 1.0;
   DATA[1019,18] := 1.0;
   DATA[1019,19] := 1.0;
   DATA[1019,20] := 148.808;
   DATA[1019,21] := 155.0115;
   DATA[1019,22] := 1.715567;
   DATA[1019,23] := 904.8449;
   DATA[1019,24] := 2.0;
   DATA[1019,25] := 2.0;
   DATA[1019,26] := 7.87798;
   DATA[1019,27] := 144.0913;
   DATA[1019,28] := 263.1056;
   DATA[1019,29] := 12.03538;
   DATA[1019,30] := 1.72443;
   DATA[1019,31] := 1.265531;
   DATA[1019,32] := 0.7351407;
   DATA[1019,33] := 0.3083624;
   DATA[1019,34] := 2.0;
   DATA[1019,35] := 250.1442;
   DATA[1019,36] := 1.649953;
   DATA[1019,37] := 189.0541;
   DATA[1019,38] := 0.000128152;
   DATA[1019,39] := 1.0;
   DATA[1020,0] := 2.541075;
   DATA[1020,1] := 665.4913;
   DATA[1020,2] := 2.0;
   DATA[1020,3] := 1.0;
   DATA[1020,4] := 262.5288;
   DATA[1020,5] := 8.462126;
   DATA[1020,6] := 315.9959;
   DATA[1020,8] := 1.0;
   DATA[1020,9] := 1.0;
   DATA[1020,10] := 1.0;
   DATA[1020,11] := 2.010372;
   DATA[1020,13] := 1011.279;
   DATA[1020,14] := 1.0;
   DATA[1020,15] := 1.0;
   DATA[1020,16] := 1.0;
   DATA[1020,17] := 1.0;
   DATA[1020,18] := 1.0;
   DATA[1020,19] := 1.0;
   DATA[1020,20] := 148.808;
   DATA[1020,21] := 155.0115;
   DATA[1020,22] := 1.713645;
   DATA[1020,23] := 904.3835;
   DATA[1020,24] := 2.0;
   DATA[1020,25] := 2.0;
   DATA[1020,26] := 7.87798;
   DATA[1020,27] := 144.0913;
   DATA[1020,28] := 263.1056;
   DATA[1020,29] := 12.03538;
   DATA[1020,30] := 1.72443;
   DATA[1020,31] := 1.28436;
   DATA[1020,32] := 0.7351407;
   DATA[1020,33] := 0.3083624;
   DATA[1020,34] := 2.0;
   DATA[1020,35] := 250.1442;
   DATA[1020,36] := 1.665972;
   DATA[1020,37] := 189.0541;
   DATA[1020,38] := 0.000128152;
   DATA[1020,39] := 1.0;
   DATA[1021,0] := 2.542356;
   DATA[1021,1] := 666.4333;
   DATA[1021,2] := 2.0;
   DATA[1021,3] := 1.0;
   DATA[1021,4] := 262.5288;
   DATA[1021,5] := 8.462126;
   DATA[1021,6] := 315.8165;
   DATA[1021,8] := 1.0;
   DATA[1021,9] := 1.0;
   DATA[1021,10] := 1.0;
   DATA[1021,11] := 2.010372;
   DATA[1021,13] := 1011.279;
   DATA[1021,14] := 1.0;
   DATA[1021,15] := 1.0;
   DATA[1021,16] := 1.0;
   DATA[1021,17] := 1.0;
   DATA[1021,18] := 1.0;
   DATA[1021,19] := 1.0;
   DATA[1021,20] := 148.808;
   DATA[1021,21] := 155.0115;
   DATA[1021,22] := 1.713645;
   DATA[1021,23] := 903.8452;
   DATA[1021,24] := 2.0;
   DATA[1021,25] := 2.0;
   DATA[1021,26] := 7.87798;
   DATA[1021,27] := 144.0913;
   DATA[1021,28] := 263.1056;
   DATA[1021,29] := 12.03538;
   DATA[1021,30] := 1.72443;
   DATA[1021,31] := 1.292174;
   DATA[1021,32] := 0.7351407;
   DATA[1021,33] := 0.3083624;
   DATA[1021,34] := 2.0;
   DATA[1021,35] := 250.4005;
   DATA[1021,36] := 1.665972;
   DATA[1021,37] := 189.0541;
   DATA[1021,38] := 0.000128152;
   DATA[1021,39] := 1.0;
   DATA[1022,0] := 2.54588;
   DATA[1022,1] := 666.5511;
   DATA[1022,2] := 2.0;
   DATA[1022,3] := 1.0;
   DATA[1022,4] := 262.5288;
   DATA[1022,5] := 8.462126;
   DATA[1022,6] := 315.8165;
   DATA[1022,8] := 1.0;
   DATA[1022,9] := 1.0;
   DATA[1022,10] := 1.0;
   DATA[1022,11] := 2.010372;
   DATA[1022,13] := 1011.119;
   DATA[1022,14] := 1.0;
   DATA[1022,15] := 1.0;
   DATA[1022,16] := 1.0;
   DATA[1022,17] := 1.0;
   DATA[1022,18] := 1.0;
   DATA[1022,19] := 1.0;
   DATA[1022,20] := 148.808;
   DATA[1022,21] := 155.0115;
   DATA[1022,22] := 1.713645;
   DATA[1022,23] := 903.6913;
   DATA[1022,24] := 2.0;
   DATA[1022,25] := 2.0;
   DATA[1022,26] := 7.87798;
   DATA[1022,27] := 144.0913;
   DATA[1022,28] := 263.1056;
   DATA[1022,29] := 12.03538;
   DATA[1022,30] := 1.72443;
   DATA[1022,31] := 1.292174;
   DATA[1022,32] := 0.7351407;
   DATA[1022,33] := 0.3083624;
   DATA[1022,34] := 2.0;
   DATA[1022,35] := 250.4005;
   DATA[1022,36] := 1.69801;
   DATA[1022,37] := 189.1823;
   DATA[1022,38] := 0.000128152;
   DATA[1022,39] := 1.0;
   DATA[1023,0] := 2.54588;
   DATA[1023,1] := 667.3361;
   DATA[1023,2] := 2.0;
   DATA[1023,3] := 1.0;
   DATA[1023,4] := 262.5288;
   DATA[1023,5] := 8.462126;
   DATA[1023,6] := 315.8165;
   DATA[1023,8] := 1.0;
   DATA[1023,9] := 1.0;
   DATA[1023,10] := 1.0;
   DATA[1023,11] := 2.010372;
   DATA[1023,13] := 1011.239;
   DATA[1023,14] := 1.0;
   DATA[1023,15] := 1.0;
   DATA[1023,16] := 1.0;
   DATA[1023,17] := 1.0;
   DATA[1023,18] := 1.0;
   DATA[1023,19] := 1.0;
   DATA[1023,20] := 148.808;
   DATA[1023,21] := 155.0115;
   DATA[1023,22] := 1.716592;
   DATA[1023,23] := 903.2299;
   DATA[1023,24] := 2.0;
   DATA[1023,25] := 2.0;
   DATA[1023,26] := 7.87798;
   DATA[1023,27] := 144.0913;
   DATA[1023,28] := 263.1056;
   DATA[1023,29] := 12.03538;
   DATA[1023,30] := 1.728531;
   DATA[1023,31] := 1.292174;
   DATA[1023,32] := 0.7351407;
   DATA[1023,33] := 0.3083624;
   DATA[1023,34] := 2.0;
   DATA[1023,35] := 250.5608;
   DATA[1023,36] := 1.730048;
   DATA[1023,37] := 189.3425;
   DATA[1023,38] := 0.000128152;
   DATA[1023,39] := 1.0;
   DATA[1024,0] := 2.54588;
   DATA[1024,1] := 667.6894;
   DATA[1024,2] := 2.0;
   DATA[1024,3] := 1.0;
   DATA[1024,4] := 262.5288;
   DATA[1024,5] := 8.462126;
   DATA[1024,6] := 315.9446;
   DATA[1024,8] := 1.0;
   DATA[1024,9] := 1.0;
   DATA[1024,10] := 1.0;
   DATA[1024,11] := 2.010372;
   DATA[1024,13] := 1011.56;
   DATA[1024,14] := 1.0;
   DATA[1024,15] := 1.0;
   DATA[1024,16] := 1.0;
   DATA[1024,17] := 1.0;
   DATA[1024,18] := 1.0;
   DATA[1024,19] := 1.0;
   DATA[1024,20] := 148.808;
   DATA[1024,21] := 154.8065;
   DATA[1024,22] := 1.717746;
   DATA[1024,23] := 903.0761;
   DATA[1024,24] := 2.0;
   DATA[1024,25] := 2.0;
   DATA[1024,26] := 7.87798;
   DATA[1024,27] := 144.0913;
   DATA[1024,28] := 263.1056;
   DATA[1024,29] := 12.03538;
   DATA[1024,30] := 1.728531;
   DATA[1024,31] := 1.292174;
   DATA[1024,32] := 0.7351407;
   DATA[1024,33] := 0.3071454;
   DATA[1024,34] := 2.0;
   DATA[1024,35] := 250.5608;
   DATA[1024,36] := 1.730048;
   DATA[1024,37] := 189.3425;
   DATA[1024,38] := 0.000128152;
   DATA[1024,39] := 1.0;
   DATA[1025,0] := 2.54588;
   DATA[1025,1] := 667.6501;
   DATA[1025,2] := 2.0;
   DATA[1025,3] := 1.0;
   DATA[1025,4] := 262.5288;
   DATA[1025,5] := 8.462126;
   DATA[1025,6] := 315.9446;
   DATA[1025,8] := 1.0;
   DATA[1025,9] := 1.0;
   DATA[1025,10] := 1.0;
   DATA[1025,11] := 2.010372;
   DATA[1025,13] := 1011.56;
   DATA[1025,14] := 1.0;
   DATA[1025,15] := 1.0;
   DATA[1025,16] := 1.0;
   DATA[1025,17] := 1.0;
   DATA[1025,18] := 1.0;
   DATA[1025,19] := 1.0;
   DATA[1025,20] := 148.808;
   DATA[1025,21] := 154.8065;
   DATA[1025,22] := 1.717746;
   DATA[1025,23] := 902.4609;
   DATA[1025,24] := 2.0;
   DATA[1025,25] := 2.0;
   DATA[1025,26] := 7.87798;
   DATA[1025,27] := 144.0913;
   DATA[1025,28] := 263.1056;
   DATA[1025,29] := 12.03538;
   DATA[1025,30] := 1.726865;
   DATA[1025,31] := 1.292174;
   DATA[1025,32] := 0.7351407;
   DATA[1025,33] := 0.3068891;
   DATA[1025,34] := 2.0;
   DATA[1025,35] := 250.5608;
   DATA[1025,36] := 1.730048;
   DATA[1025,37] := 189.3425;
   DATA[1025,38] := 0.000128152;
   DATA[1025,39] := 1.0;
   DATA[1026,0] := 2.54588;
   DATA[1026,1] := 668.1997;
   DATA[1026,2] := 2.0;
   DATA[1026,3] := 1.0;
   DATA[1026,4] := 262.5288;
   DATA[1026,5] := 8.46501;
   DATA[1026,6] := 315.9446;
   DATA[1026,8] := 1.0;
   DATA[1026,9] := 1.0;
   DATA[1026,10] := 1.0;
   DATA[1026,11] := 2.010372;
   DATA[1026,13] := 1011.159;
   DATA[1026,14] := 1.0;
   DATA[1026,15] := 1.0;
   DATA[1026,16] := 1.0;
   DATA[1026,17] := 1.0;
   DATA[1026,18] := 1.0;
   DATA[1026,19] := 1.0;
   DATA[1026,20] := 148.808;
   DATA[1026,21] := 154.8065;
   DATA[1026,22] := 1.717746;
   DATA[1026,23] := 901.7688;
   DATA[1026,24] := 2.0;
   DATA[1026,25] := 2.0;
   DATA[1026,26] := 7.87798;
   DATA[1026,27] := 144.0913;
   DATA[1026,28] := 263.1056;
   DATA[1026,29] := 12.03538;
   DATA[1026,30] := 1.726224;
   DATA[1026,31] := 1.300243;
   DATA[1026,32] := 0.7351407;
   DATA[1026,33] := 0.3068891;
   DATA[1026,34] := 2.0;
   DATA[1026,35] := 250.721;
   DATA[1026,36] := 1.730048;
   DATA[1026,37] := 189.3425;
   DATA[1026,38] := 0.000128152;
   DATA[1026,39] := 1.0;
   DATA[1027,0] := 2.539474;
   DATA[1027,1] := 668.3174;
   DATA[1027,2] := 2.0;
   DATA[1027,3] := 1.0;
   DATA[1027,4] := 262.5288;
   DATA[1027,5] := 8.46501;
   DATA[1027,6] := 315.9446;
   DATA[1027,8] := 1.0;
   DATA[1027,9] := 1.0;
   DATA[1027,10] := 1.0;
   DATA[1027,11] := 2.010372;
   DATA[1027,13] := 1010.959;
   DATA[1027,14] := 1.0;
   DATA[1027,15] := 1.0;
   DATA[1027,16] := 1.0;
   DATA[1027,17] := 1.0;
   DATA[1027,18] := 1.0;
   DATA[1027,19] := 1.0;
   DATA[1027,20] := 148.808;
   DATA[1027,21] := 154.8065;
   DATA[1027,22] := 1.718643;
   DATA[1027,23] := 901.1536;
   DATA[1027,24] := 2.0;
   DATA[1027,25] := 2.0;
   DATA[1027,26] := 7.87798;
   DATA[1027,27] := 144.0913;
   DATA[1027,28] := 263.1056;
   DATA[1027,29] := 12.03538;
   DATA[1027,30] := 1.726224;
   DATA[1027,31] := 1.296657;
   DATA[1027,32] := 0.7351407;
   DATA[1027,33] := 0.3068891;
   DATA[1027,34] := 2.0;
   DATA[1027,35] := 250.753;
   DATA[1027,36] := 1.730048;
   DATA[1027,37] := 189.3425;
   DATA[1027,38] := 0.000128152;
   DATA[1027,39] := 1.0;
   DATA[1028,0] := 2.536912;
   DATA[1028,1] := 668.239;
   DATA[1028,2] := 2.0;
   DATA[1028,3] := 1.0;
   DATA[1028,4] := 262.5288;
   DATA[1028,5] := 8.46501;
   DATA[1028,6] := 315.9446;
   DATA[1028,8] := 1.0;
   DATA[1028,9] := 1.0;
   DATA[1028,10] := 1.0;
   DATA[1028,11] := 2.010372;
   DATA[1028,13] := 1011.039;
   DATA[1028,14] := 1.0;
   DATA[1028,15] := 1.0;
   DATA[1028,16] := 1.0;
   DATA[1028,17] := 1.0;
   DATA[1028,18] := 1.0;
   DATA[1028,19] := 1.0;
   DATA[1028,20] := 148.808;
   DATA[1028,21] := 154.8065;
   DATA[1028,22] := 1.720437;
   DATA[1028,23] := 901.0382;
   DATA[1028,24] := 2.0;
   DATA[1028,25] := 2.0;
   DATA[1028,26] := 7.87798;
   DATA[1028,27] := 144.0913;
   DATA[1028,28] := 263.1056;
   DATA[1028,29] := 12.03538;
   DATA[1028,30] := 1.726224;
   DATA[1028,31] := 1.291918;
   DATA[1028,32] := 0.7351407;
   DATA[1028,33] := 0.3068891;
   DATA[1028,34] := 2.0;
   DATA[1028,35] := 250.8011;
   DATA[1028,36] := 1.730048;
   DATA[1028,37] := 189.4867;
   DATA[1028,38] := 0.000128152;
   DATA[1028,39] := 1.0;
   DATA[1029,0] := 2.532428;
   DATA[1029,1] := 668.5137;
   DATA[1029,2] := 2.0;
   DATA[1029,3] := 1.0;
   DATA[1029,4] := 262.5288;
   DATA[1029,5] := 8.46501;
   DATA[1029,6] := 315.9446;
   DATA[1029,8] := 1.0;
   DATA[1029,9] := 1.0;
   DATA[1029,10] := 1.0;
   DATA[1029,11] := 2.010372;
   DATA[1029,13] := 1010.879;
   DATA[1029,14] := 1.0;
   DATA[1029,15] := 1.0;
   DATA[1029,16] := 1.0;
   DATA[1029,17] := 1.0;
   DATA[1029,18] := 1.0;
   DATA[1029,19] := 1.0;
   DATA[1029,20] := 148.808;
   DATA[1029,21] := 154.8065;
   DATA[1029,22] := 1.720565;
   DATA[1029,23] := 900.0769;
   DATA[1029,24] := 2.0;
   DATA[1029,25] := 2.0;
   DATA[1029,26] := 7.87798;
   DATA[1029,27] := 144.0913;
   DATA[1029,28] := 263.1056;
   DATA[1029,29] := 12.03538;
   DATA[1029,30] := 1.727634;
   DATA[1029,31] := 1.282311;
   DATA[1029,32] := 0.7351407;
   DATA[1029,33] := 0.3065689;
   DATA[1029,34] := 2.0;
   DATA[1029,35] := 250.8011;
   DATA[1029,36] := 1.730048;
   DATA[1029,37] := 189.5187;
   DATA[1029,38] := 0.000128152;
   DATA[1029,39] := 1.0;
   DATA[1030,0] := 2.532428;
   DATA[1030,1] := 669.2203;
   DATA[1030,2] := 2.0;
   DATA[1030,3] := 1.0;
   DATA[1030,4] := 262.5288;
   DATA[1030,5] := 8.46501;
   DATA[1030,6] := 315.9446;
   DATA[1030,8] := 1.0;
   DATA[1030,9] := 1.0;
   DATA[1030,10] := 1.0;
   DATA[1030,11] := 2.010372;
   DATA[1030,13] := 1010.879;
   DATA[1030,14] := 1.0;
   DATA[1030,15] := 1.0;
   DATA[1030,16] := 1.0;
   DATA[1030,17] := 1.0;
   DATA[1030,18] := 1.0;
   DATA[1030,19] := 1.0;
   DATA[1030,20] := 148.808;
   DATA[1030,21] := 154.6526;
   DATA[1030,22] := 1.720565;
   DATA[1030,23] := 899.5001;
   DATA[1030,24] := 2.0;
   DATA[1030,25] := 2.0;
   DATA[1030,26] := 7.87798;
   DATA[1030,27] := 144.0913;
   DATA[1030,28] := 263.1056;
   DATA[1030,29] := 12.03538;
   DATA[1030,30] := 1.727634;
   DATA[1030,31] := 1.281927;
   DATA[1030,32] := 0.7351407;
   DATA[1030,33] := 0.3065689;
   DATA[1030,34] := 2.0;
   DATA[1030,35] := 250.8011;
   DATA[1030,36] := 1.730048;
   DATA[1030,37] := 189.6148;
   DATA[1030,38] := 0.000128152;
   DATA[1030,39] := 1.0;
   DATA[1031,0] := 2.532428;
   DATA[1031,1] := 669.5735;
   DATA[1031,2] := 2.0;
   DATA[1031,3] := 1.0;
   DATA[1031,4] := 262.5288;
   DATA[1031,5] := 8.464048;
   DATA[1031,6] := 315.9446;
   DATA[1031,8] := 1.0;
   DATA[1031,9] := 1.0;
   DATA[1031,10] := 1.0;
   DATA[1031,11] := 2.010372;
   DATA[1031,13] := 1010.959;
   DATA[1031,14] := 1.0;
   DATA[1031,15] := 1.0;
   DATA[1031,16] := 1.0;
   DATA[1031,17] := 1.0;
   DATA[1031,18] := 1.0;
   DATA[1031,19] := 1.0;
   DATA[1031,20] := 148.808;
   DATA[1031,21] := 154.6526;
   DATA[1031,22] := 1.720565;
   DATA[1031,23] := 899.2694;
   DATA[1031,24] := 2.0;
   DATA[1031,25] := 2.0;
   DATA[1031,26] := 7.87798;
   DATA[1031,27] := 144.0913;
   DATA[1031,28] := 263.1056;
   DATA[1031,29] := 12.03538;
   DATA[1031,30] := 1.727634;
   DATA[1031,31] := 1.286922;
   DATA[1031,32] := 0.7351407;
   DATA[1031,33] := 0.3065689;
   DATA[1031,34] := 2.0;
   DATA[1031,35] := 250.8011;
   DATA[1031,36] := 1.730048;
   DATA[1031,37] := 189.6148;
   DATA[1031,38] := 0.000128152;
   DATA[1031,39] := 1.0;
   DATA[1032,0] := 2.538513;
   DATA[1032,1] := 669.652;
   DATA[1032,2] := 2.0;
   DATA[1032,3] := 1.0;
   DATA[1032,4] := 262.5288;
   DATA[1032,5] := 8.462446;
   DATA[1032,6] := 316.0728;
   DATA[1032,8] := 1.0;
   DATA[1032,9] := 1.0;
   DATA[1032,10] := 1.0;
   DATA[1032,11] := 2.010372;
   DATA[1032,13] := 1011.079;
   DATA[1032,14] := 1.0;
   DATA[1032,15] := 1.0;
   DATA[1032,16] := 1.0;
   DATA[1032,17] := 1.0;
   DATA[1032,18] := 1.0;
   DATA[1032,19] := 1.0;
   DATA[1032,20] := 148.808;
   DATA[1032,21] := 154.6526;
   DATA[1032,22] := 1.719668;
   DATA[1032,23] := 899.0002;
   DATA[1032,24] := 2.0;
   DATA[1032,25] := 2.0;
   DATA[1032,26] := 7.87798;
   DATA[1032,27] := 144.0913;
   DATA[1032,28] := 263.1056;
   DATA[1032,29] := 12.03538;
   DATA[1032,30] := 1.727634;
   DATA[1032,31] := 1.29243;
   DATA[1032,32] := 0.7351407;
   DATA[1032,33] := 0.3065689;
   DATA[1032,34] := 2.0;
   DATA[1032,35] := 250.8652;
   DATA[1032,36] := 1.730048;
   DATA[1032,37] := 189.6148;
   DATA[1032,38] := 0.000128152;
   DATA[1032,39] := 1.0;
   DATA[1033,0] := 2.543638;
   DATA[1033,1] := 670.0839;
   DATA[1033,2] := 2.0;
   DATA[1033,3] := 1.0;
   DATA[1033,4] := 262.5288;
   DATA[1033,5] := 8.461164;
   DATA[1033,6] := 316.0728;
   DATA[1033,8] := 1.0;
   DATA[1033,9] := 1.0;
   DATA[1033,10] := 1.0;
   DATA[1033,11] := 2.010372;
   DATA[1033,13] := 1010.959;
   DATA[1033,14] := 1.0;
   DATA[1033,15] := 1.0;
   DATA[1033,16] := 1.0;
   DATA[1033,17] := 1.0;
   DATA[1033,18] := 1.0;
   DATA[1033,19] := 1.0;
   DATA[1033,20] := 148.808;
   DATA[1033,21] := 154.6526;
   DATA[1033,22] := 1.718643;
   DATA[1033,23] := 898.4619;
   DATA[1033,24] := 2.0;
   DATA[1033,25] := 2.0;
   DATA[1033,26] := 7.87798;
   DATA[1033,27] := 144.0913;
   DATA[1033,28] := 263.1056;
   DATA[1033,29] := 12.03538;
   DATA[1033,30] := 1.72789;
   DATA[1033,31] := 1.29243;
   DATA[1033,32] := 0.7351407;
   DATA[1033,33] := 0.3065689;
   DATA[1033,34] := 2.0;
   DATA[1033,35] := 250.9453;
   DATA[1033,36] := 1.730048;
   DATA[1033,37] := 189.6148;
   DATA[1033,38] := 0.000128152;
   DATA[1033,39] := 1.0;
   DATA[1034,0] := 2.54684;
   DATA[1034,1] := 671.1437;
   DATA[1034,2] := 2.0;
   DATA[1034,3] := 1.0;
   DATA[1034,4] := 262.5288;
   DATA[1034,5] := 8.461164;
   DATA[1034,6] := 316.0728;
   DATA[1034,8] := 1.0;
   DATA[1034,9] := 1.0;
   DATA[1034,10] := 1.0;
   DATA[1034,11] := 2.010372;
   DATA[1034,13] := 1011.039;
   DATA[1034,14] := 1.0;
   DATA[1034,15] := 1.0;
   DATA[1034,16] := 1.0;
   DATA[1034,17] := 1.0;
   DATA[1034,18] := 1.0;
   DATA[1034,19] := 1.0;
   DATA[1034,20] := 148.808;
   DATA[1034,21] := 154.8321;
   DATA[1034,22] := 1.718643;
   DATA[1034,23] := 898.0389;
   DATA[1034,24] := 2.0;
   DATA[1034,25] := 2.0;
   DATA[1034,26] := 7.87798;
   DATA[1034,27] := 144.0913;
   DATA[1034,28] := 263.1056;
   DATA[1034,29] := 12.03538;
   DATA[1034,30] := 1.728788;
   DATA[1034,31] := 1.283592;
   DATA[1034,32] := 0.7351407;
   DATA[1034,33] := 0.3065689;
   DATA[1034,34] := 2.0;
   DATA[1034,35] := 250.9453;
   DATA[1034,36] := 1.730048;
   DATA[1034,37] := 189.6148;
   DATA[1034,38] := 0.000128152;
   DATA[1034,39] := 1.0;
   DATA[1035,0] := 2.54684;
   DATA[1035,1] := 671.811;
   DATA[1035,2] := 2.0;
   DATA[1035,3] := 1.0;
   DATA[1035,4] := 262.5288;
   DATA[1035,5] := 8.461164;
   DATA[1035,6] := 316.0728;
   DATA[1035,8] := 1.0;
   DATA[1035,9] := 1.0;
   DATA[1035,10] := 1.0;
   DATA[1035,11] := 2.010372;
   DATA[1035,13] := 1010.919;
   DATA[1035,14] := 1.0;
   DATA[1035,15] := 1.0;
   DATA[1035,16] := 1.0;
   DATA[1035,17] := 1.0;
   DATA[1035,18] := 1.0;
   DATA[1035,19] := 1.0;
   DATA[1035,20] := 148.808;
   DATA[1035,21] := 154.8321;
   DATA[1035,22] := 1.719796;
   DATA[1035,23] := 897.8467;
   DATA[1035,24] := 2.0;
   DATA[1035,25] := 2.0;
   DATA[1035,26] := 7.87798;
   DATA[1035,27] := 144.0913;
   DATA[1035,28] := 263.1056;
   DATA[1035,29] := 12.03538;
   DATA[1035,30] := 1.729428;
   DATA[1035,31] := 1.264506;
   DATA[1035,32] := 0.7351407;
   DATA[1035,33] := 0.3065689;
   DATA[1035,34] := 2.0;
   DATA[1035,35] := 250.9453;
   DATA[1035,36] := 1.730048;
   DATA[1035,37] := 189.6148;
   DATA[1035,38] := 0.000128152;
   DATA[1035,39] := 1.0;
   DATA[1036,0] := 2.550684;
   DATA[1036,1] := 672.125;
   DATA[1036,2] := 2.0;
   DATA[1036,3] := 1.0;
   DATA[1036,4] := 262.5288;
   DATA[1036,5] := 8.461164;
   DATA[1036,6] := 316.0728;
   DATA[1036,8] := 1.0;
   DATA[1036,9] := 1.0;
   DATA[1036,10] := 1.0;
   DATA[1036,11] := 2.010372;
   DATA[1036,13] := 1010.718;
   DATA[1036,14] := 1.0;
   DATA[1036,15] := 1.0;
   DATA[1036,16] := 1.0;
   DATA[1036,17] := 1.0;
   DATA[1036,18] := 1.0;
   DATA[1036,19] := 1.0;
   DATA[1036,20] := 148.808;
   DATA[1036,21] := 154.8321;
   DATA[1036,22] := 1.719796;
   DATA[1036,23] := 897.616;
   DATA[1036,24] := 2.0;
   DATA[1036,25] := 2.0;
   DATA[1036,26] := 7.87798;
   DATA[1036,27] := 144.0913;
   DATA[1036,28] := 263.1056;
   DATA[1036,29] := 12.03538;
   DATA[1036,30] := 1.729428;
   DATA[1036,31] := 1.262457;
   DATA[1036,32] := 0.7351407;
   DATA[1036,33] := 0.3065689;
   DATA[1036,34] := 2.0;
   DATA[1036,35] := 250.9453;
   DATA[1036,36] := 1.730048;
   DATA[1036,37] := 189.6148;
   DATA[1036,38] := 0.000128152;
   DATA[1036,39] := 1.0;
   DATA[1037,0] := 2.550684;
   DATA[1037,1] := 673.0278;
   DATA[1037,2] := 2.0;
   DATA[1037,3] := 1.0;
   DATA[1037,4] := 262.5288;
   DATA[1037,5] := 8.461164;
   DATA[1037,6] := 316.201;
   DATA[1037,8] := 1.0;
   DATA[1037,9] := 1.0;
   DATA[1037,10] := 1.0;
   DATA[1037,11] := 2.010372;
   DATA[1037,13] := 1011.279;
   DATA[1037,14] := 1.0;
   DATA[1037,15] := 1.0;
   DATA[1037,16] := 1.0;
   DATA[1037,17] := 1.0;
   DATA[1037,18] := 1.0;
   DATA[1037,19] := 1.0;
   DATA[1037,20] := 148.808;
   DATA[1037,21] := 154.8321;
   DATA[1037,22] := 1.719796;
   DATA[1037,23] := 897.27;
   DATA[1037,24] := 2.0;
   DATA[1037,25] := 2.0;
   DATA[1037,26] := 7.87798;
   DATA[1037,27] := 144.0913;
   DATA[1037,28] := 263.1056;
   DATA[1037,29] := 12.03538;
   DATA[1037,30] := 1.729428;
   DATA[1037,31] := 1.265147;
   DATA[1037,32] := 0.7351407;
   DATA[1037,33] := 0.3080421;
   DATA[1037,34] := 2.0;
   DATA[1037,35] := 250.753;
   DATA[1037,36] := 1.730048;
   DATA[1037,37] := 189.6148;
   DATA[1037,38] := 0.000128152;
   DATA[1037,39] := 1.0;
   DATA[1038,0] := 2.550684;
   DATA[1038,1] := 673.7343;
   DATA[1038,2] := 2.0;
   DATA[1038,3] := 1.0;
   DATA[1038,4] := 262.5288;
   DATA[1038,5] := 8.463408;
   DATA[1038,6] := 316.201;
   DATA[1038,8] := 1.0;
   DATA[1038,9] := 1.0;
   DATA[1038,10] := 1.0;
   DATA[1038,11] := 2.010372;
   DATA[1038,13] := 1011.159;
   DATA[1038,14] := 1.0;
   DATA[1038,15] := 1.0;
   DATA[1038,16] := 1.0;
   DATA[1038,17] := 1.0;
   DATA[1038,18] := 1.0;
   DATA[1038,19] := 1.0;
   DATA[1038,20] := 148.808;
   DATA[1038,21] := 154.8321;
   DATA[1038,22] := 1.717361;
   DATA[1038,23] := 897.2315;
   DATA[1038,24] := 2.0;
   DATA[1038,25] := 2.0;
   DATA[1038,26] := 7.87798;
   DATA[1038,27] := 144.0913;
   DATA[1038,28] := 263.1056;
   DATA[1038,29] := 12.03538;
   DATA[1038,30] := 1.729428;
   DATA[1038,31] := 1.272704;
   DATA[1038,32] := 0.7351407;
   DATA[1038,33] := 0.3082983;
   DATA[1038,34] := 2.0;
   DATA[1038,35] := 250.6569;
   DATA[1038,36] := 1.730048;
   DATA[1038,37] := 189.6148;
   DATA[1038,38] := 0.000128152;
